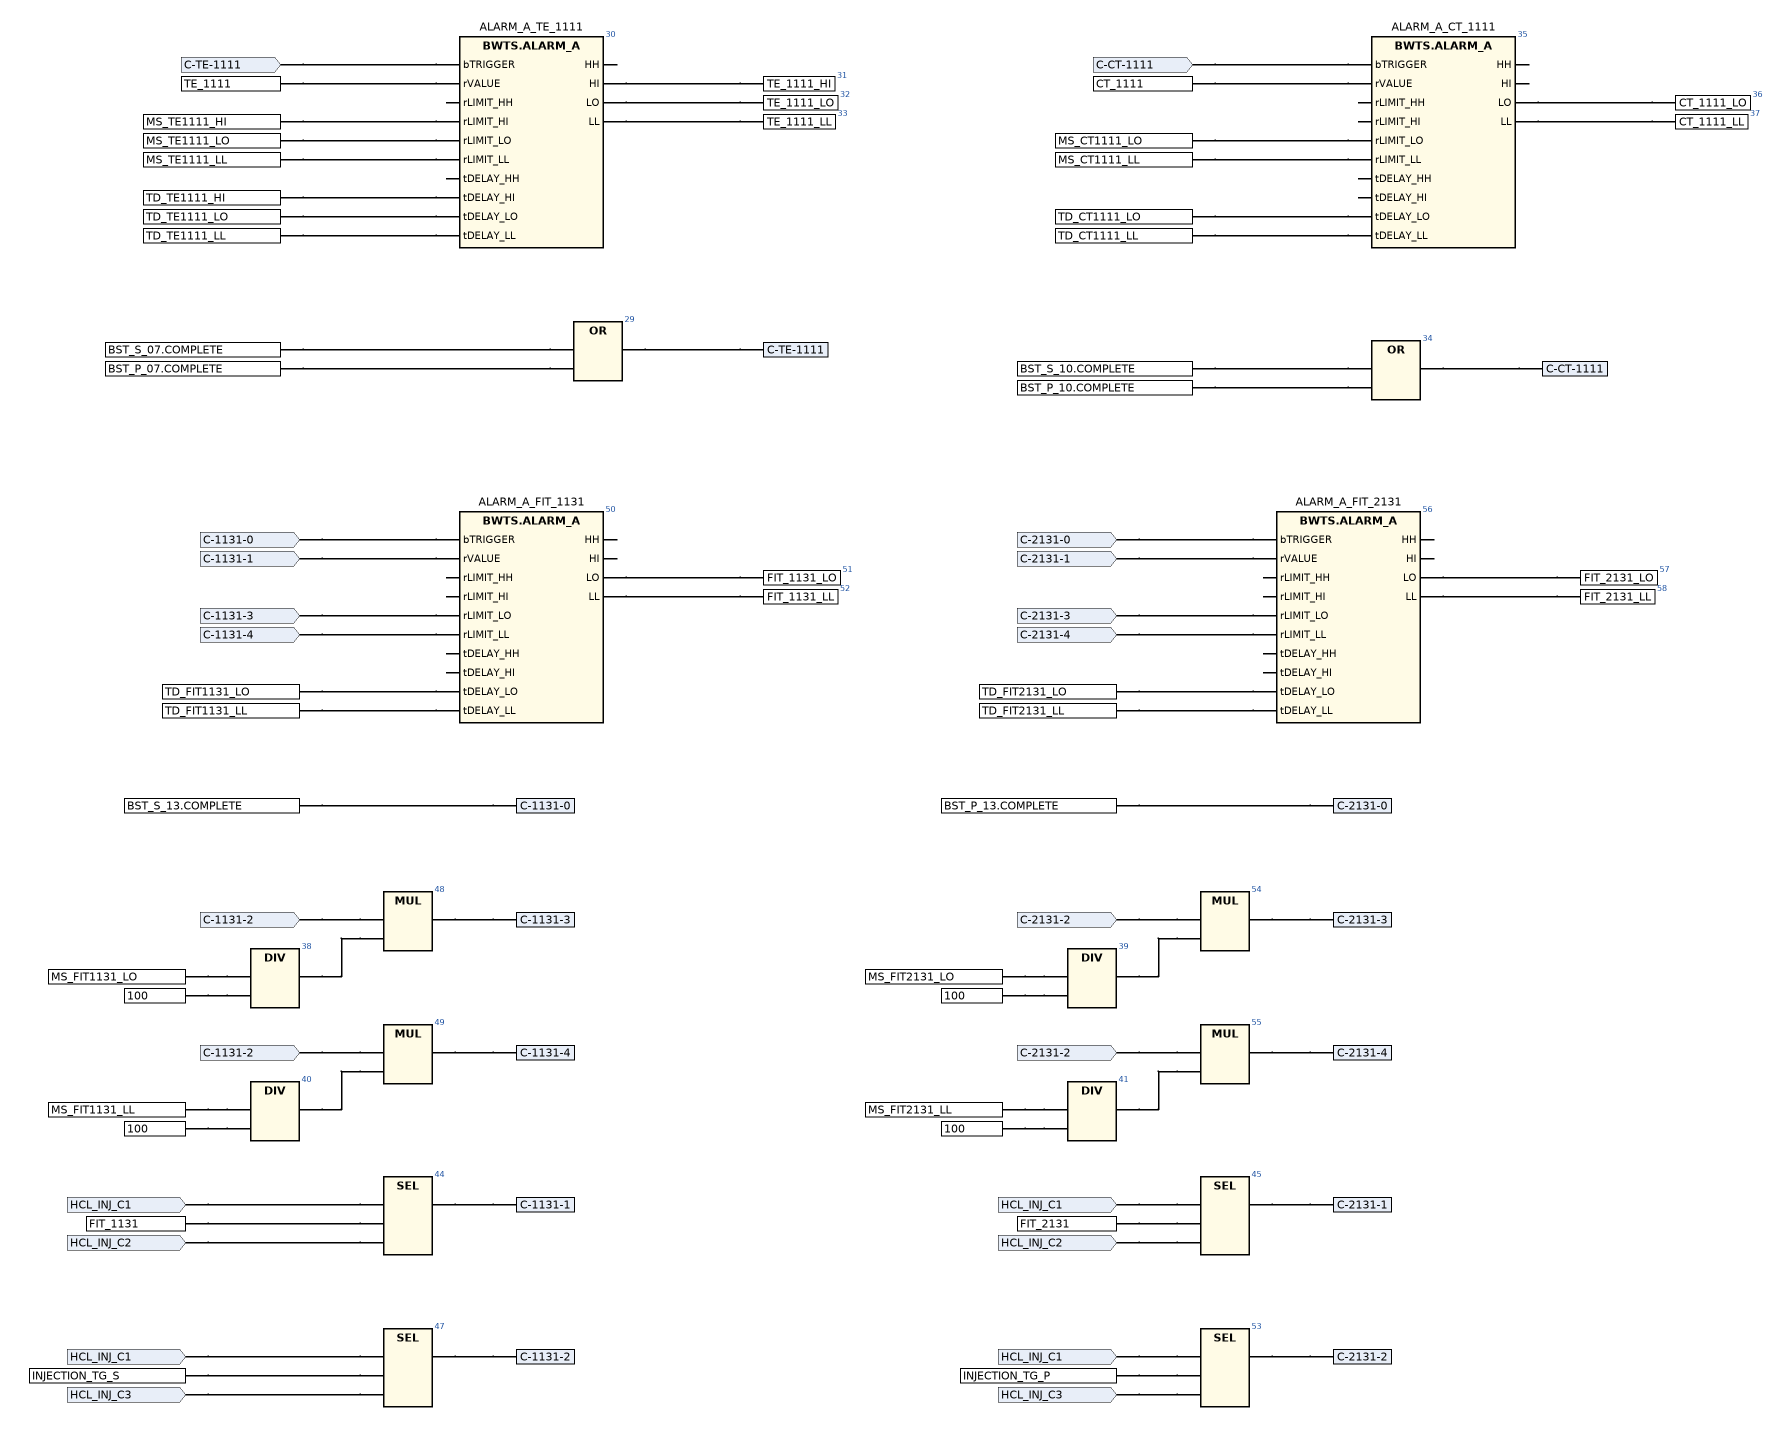
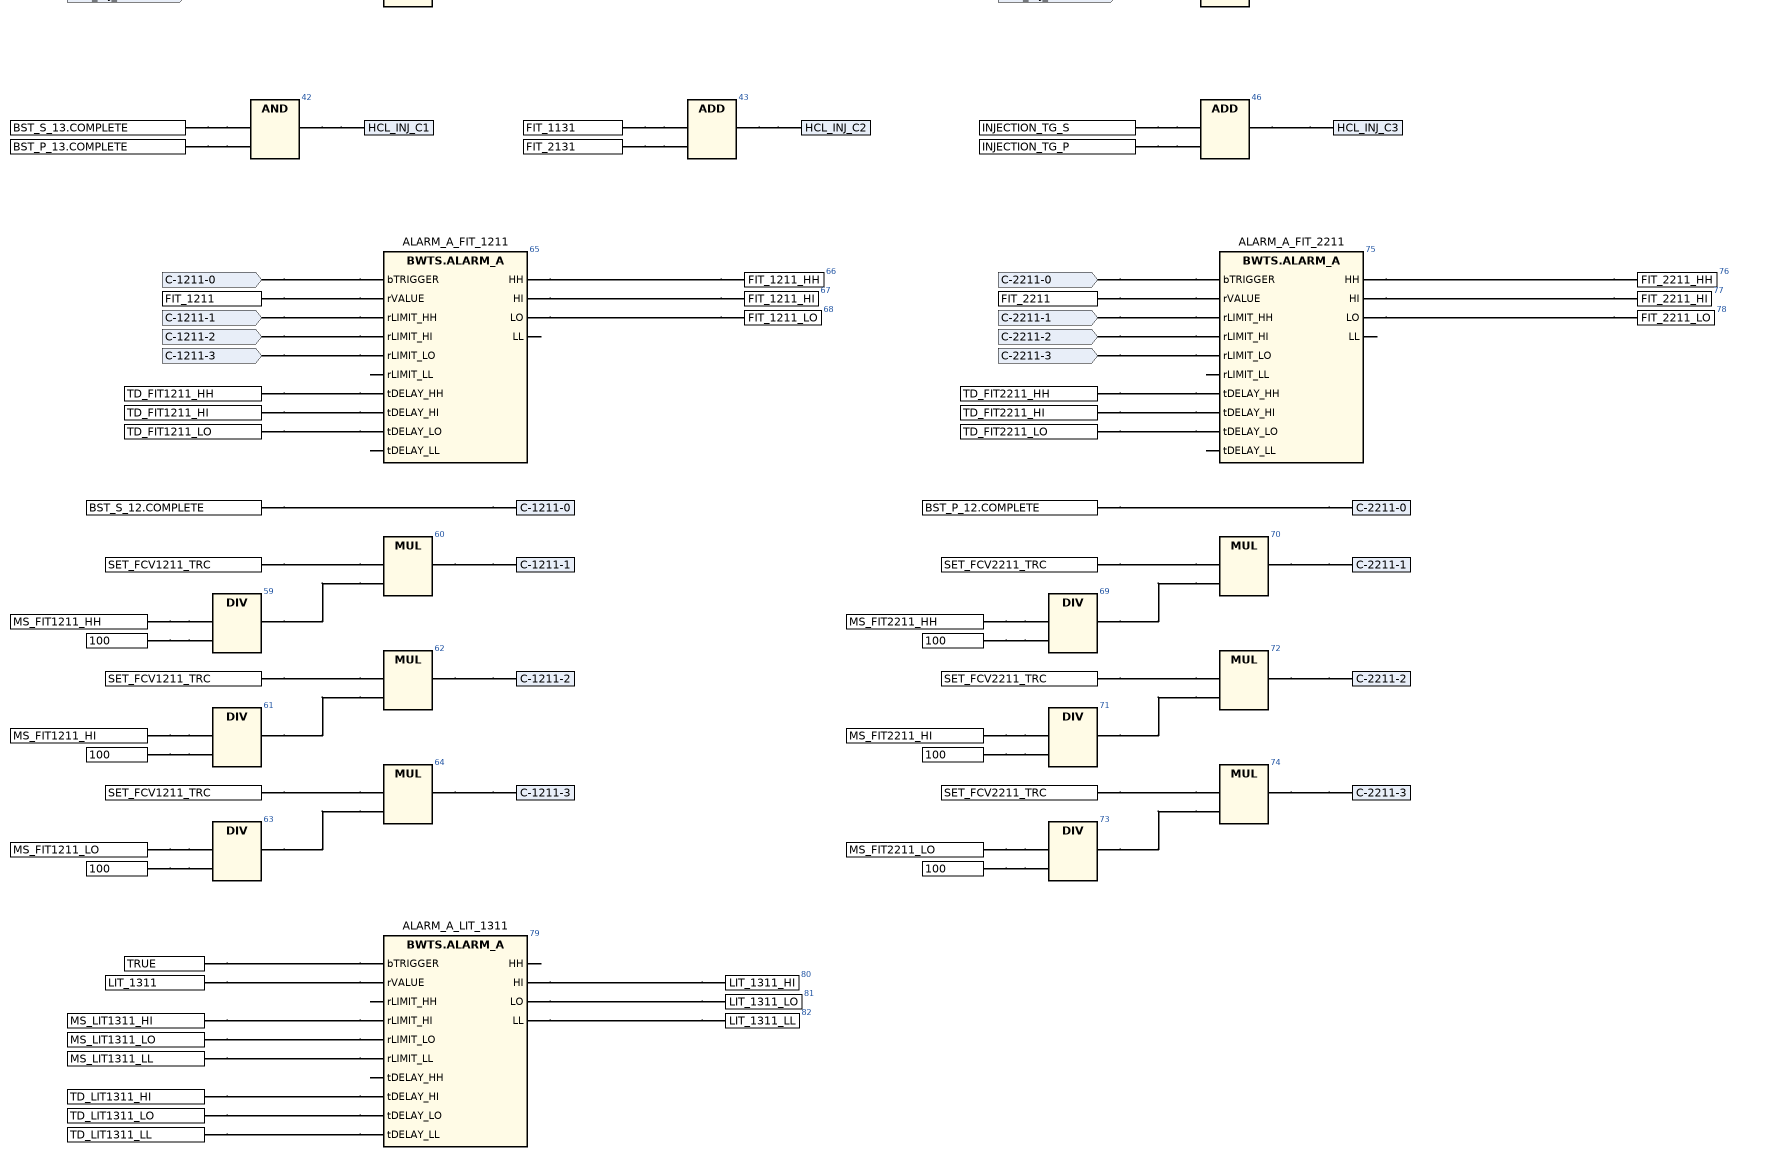
(* BST_S_06.COMPLETE OR BST_P_06.COMPLETE; result not used *)
ALARM_A_PT_1722(
    bTRIGGER := _w1,
    rVALUE := PT_1722,
    rLIMIT_HH := MS_PT1722_HH,
    rLIMIT_HI := MS_PT1722_HI,
    rLIMIT_LO := MS_PT1722_LO,
    tDELAY_HH := TD_PT1722_HH,
    tDELAY_HI := TD_PT1722_HI,
    tDELAY_LO := TD_PT1722_LO); // BWTS.ALARM_A
PT_1722_HH := ALARM_A_PT_1722.HH;
PT_1722_HI := ALARM_A_PT_1722.HI;
PT_1722_LO := ALARM_A_PT_1722.LO;
ALARM_A_PT_1721(
    bTRIGGER := _w2,
    rVALUE := PT_1721,
    rLIMIT_HI := MS_PT1721_HI,
    rLIMIT_LO := MS_PT1721_LO,
    rLIMIT_LL := MS_PT1721_LL,
    tDELAY_HI := TD_PT1721_HI,
    tDELAY_LO := TD_PT1721_LO,
    tDELAY_LL := TD_PT1721_LL); // BWTS.ALARM_A
PT_1721_HI := ALARM_A_PT_1721.HI;
PT_1721_LO := ALARM_A_PT_1721.LO;
PT_1721_LL := ALARM_A_PT_1721.LL;
ALARM_A_P_171(
    bTRIGGER := _w3,
    rVALUE := DP_P171,
    rLIMIT_HH := MS_DP171_HH,
    rLIMIT_HI := MS_DP171_HI,
    tDELAY_HH := TD_DP171_HH,
    tDELAY_HI := TD_DP171_HI); // BWTS.ALARM_A
SWFU_DP_HH := ALARM_A_P_171.HH;
SWFU_DP_HI := ALARM_A_P_171.HI;
(* BST_S_01.COMPLETE OR BST_P_01.COMPLETE; result not used *)
ALARM_A_PT_1121(
    bTRIGGER := _w4,
    rVALUE := PT_1121,
    rLIMIT_HI := MS_PT1121_HI,
    rLIMIT_LO := MS_PT1121_LO,
    rLIMIT_LL := MS_PT1121_LL,
    tDELAY_HI := TD_PT1121_HI,
    tDELAY_LO := TD_PT1121_LO,
    tDELAY_LL := TD_PT1121_LL); // BWTS.ALARM_A
PT_1121_HI := ALARM_A_PT_1121.HI;
PT_1121_LO := ALARM_A_PT_1121.LO;
PT_1121_LL := ALARM_A_PT_1121.LL;
ALARM_A_AIT_1121(
    bTRIGGER := TRUE,
    rVALUE := AIT_1121,
    rLIMIT_HH := MS_AIT1121_HH,
    rLIMIT_HI := MS_AIT1121_HI,
    tDELAY_HH := TD_AIT1121_HH,
    tDELAY_HI := TD_AIT1121_HI); // BWTS.ALARM_A
AIT_1121_HH := ALARM_A_AIT_1121.HH;
AIT_1121_HI := ALARM_A_AIT_1121.HI;
ALARM_A_AIT_1122(
    bTRIGGER := TRUE,
    rVALUE := AIT_1122,
    rLIMIT_HH := MS_AIT1122_HH,
    rLIMIT_HI := MS_AIT1122_HI,
    tDELAY_HH := TD_AIT1122_HH,
    tDELAY_HI := TD_AIT1122_HI); // BWTS.ALARM_A
AIT_1122_HH := ALARM_A_AIT_1122.HH;
AIT_1122_HI := ALARM_A_AIT_1122.HI;
ALARM_A_AIT_1123(
    bTRIGGER := TRUE,
    rVALUE := AIT_1123,
    rLIMIT_HH := MS_AIT1123_HH,
    rLIMIT_HI := MS_AIT1123_HI,
    tDELAY_HH := TD_AIT1123_HH,
    tDELAY_HI := TD_AIT1123_HI); // BWTS.ALARM_A
AIT_1123_HH := ALARM_A_AIT_1123.HH;
AIT_1123_HI := ALARM_A_AIT_1123.HI;
ALARM_A_AP_LVL_01(
    bTRIGGER := MF_APT,
    rVALUE := AP_LVL_01,
    rLIMIT_LO := MS_AP_LO,
    rLIMIT_LL := MS_AP_LL,
    tDELAY_LO := TD_AP_LO,
    tDELAY_LL := TD_AP_LL); // BWTS.ALARM_A
AP_LVL_LO := ALARM_A_AP_LVL_01.LO;
AP_LVL_LL := ALARM_A_AP_LVL_01.LL;
(* BST_S_07.COMPLETE OR BST_P_07.COMPLETE; result not used *)
ALARM_A_TE_1111(
    bTRIGGER := _w5,
    rVALUE := TE_1111,
    rLIMIT_HI := MS_TE1111_HI,
    rLIMIT_LO := MS_TE1111_LO,
    rLIMIT_LL := MS_TE1111_LL,
    tDELAY_HI := TD_TE1111_HI,
    tDELAY_LO := TD_TE1111_LO,
    tDELAY_LL := TD_TE1111_LL); // BWTS.ALARM_A
TE_1111_HI := ALARM_A_TE_1111.HI;
TE_1111_LO := ALARM_A_TE_1111.LO;
TE_1111_LL := ALARM_A_TE_1111.LL;
(* BST_S_10.COMPLETE OR BST_P_10.COMPLETE; result not used *)
ALARM_A_CT_1111(
    bTRIGGER := _w6,
    rVALUE := CT_1111,
    rLIMIT_LO := MS_CT1111_LO,
    rLIMIT_LL := MS_CT1111_LL,
    tDELAY_LO := TD_CT1111_LO,
    tDELAY_LL := TD_CT1111_LL); // BWTS.ALARM_A
CT_1111_LO := ALARM_A_CT_1111.LO;
CT_1111_LL := ALARM_A_CT_1111.LL;
_w7 := MS_FIT2131_LO / 100;
_w8 := MS_FIT2131_LL / 100;
(* BST_S_13.COMPLETE AND BST_P_13.COMPLETE; result not used *)
(* FIT_1131 + FIT_2131; result not used *)
(* SEL(_w9, FIT_1131, _w10); result not used *)
(* SEL(_w11, FIT_2131, _w12); result not used *)
(* INJECTION_TG_S + INJECTION_TG_P; result not used *)
(* SEL(_w13, INJECTION_TG_S, _w14); result not used *)
(* _w15 * (MS_FIT1131_LO / 100); result not used *)
(* _w16 * (MS_FIT1131_LL / 100); result not used *)
ALARM_A_FIT_1131(
    bTRIGGER := _w17,
    rVALUE := _w18,
    rLIMIT_LO := _w19,
    rLIMIT_LL := _w20,
    tDELAY_LO := TD_FIT1131_LO,
    tDELAY_LL := TD_FIT1131_LL); // BWTS.ALARM_A
FIT_1131_LO := ALARM_A_FIT_1131.LO;
FIT_1131_LL := ALARM_A_FIT_1131.LL;
(* SEL(_w21, INJECTION_TG_P, _w22); result not used *)
(* _w23 * _w7; result not used *)
(* _w24 * _w8; result not used *)
ALARM_A_FIT_2131(
    bTRIGGER := _w25,
    rVALUE := _w26,
    rLIMIT_LO := _w27,
    rLIMIT_LL := _w28,
    tDELAY_LO := TD_FIT2131_LO,
    tDELAY_LL := TD_FIT2131_LL); // BWTS.ALARM_A
FIT_2131_LO := ALARM_A_FIT_2131.LO;
FIT_2131_LL := ALARM_A_FIT_2131.LL;
(* SET_FCV1211_TRC * (MS_FIT1211_HH / 100); result not used *)
(* SET_FCV1211_TRC * (MS_FIT1211_HI / 100); result not used *)
(* SET_FCV1211_TRC * (MS_FIT1211_LO / 100); result not used *)
ALARM_A_FIT_1211(
    bTRIGGER := _w29,
    rVALUE := FIT_1211,
    rLIMIT_HH := _w30,
    rLIMIT_HI := _w31,
    rLIMIT_LO := _w32,
    tDELAY_HH := TD_FIT1211_HH,
    tDELAY_HI := TD_FIT1211_HI,
    tDELAY_LO := TD_FIT1211_LO); // BWTS.ALARM_A
FIT_1211_HH := ALARM_A_FIT_1211.HH;
FIT_1211_HI := ALARM_A_FIT_1211.HI;
FIT_1211_LO := ALARM_A_FIT_1211.LO;
(* SET_FCV2211_TRC * (MS_FIT2211_HH / 100); result not used *)
(* SET_FCV2211_TRC * (MS_FIT2211_HI / 100); result not used *)
(* SET_FCV2211_TRC * (MS_FIT2211_LO / 100); result not used *)
ALARM_A_FIT_2211(
    bTRIGGER := _w33,
    rVALUE := FIT_2211,
    rLIMIT_HH := _w34,
    rLIMIT_HI := _w35,
    rLIMIT_LO := _w36,
    tDELAY_HH := TD_FIT2211_HH,
    tDELAY_HI := TD_FIT2211_HI,
    tDELAY_LO := TD_FIT2211_LO); // BWTS.ALARM_A
FIT_2211_HH := ALARM_A_FIT_2211.HH;
FIT_2211_HI := ALARM_A_FIT_2211.HI;
FIT_2211_LO := ALARM_A_FIT_2211.LO;
ALARM_A_LIT_1311(
    bTRIGGER := TRUE,
    rVALUE := LIT_1311,
    rLIMIT_HI := MS_LIT1311_HI,
    rLIMIT_LO := MS_LIT1311_LO,
    rLIMIT_LL := MS_LIT1311_LL,
    tDELAY_HI := TD_LIT1311_HI,
    tDELAY_LO := TD_LIT1311_LO,
    tDELAY_LL := TD_LIT1311_LL); // BWTS.ALARM_A
LIT_1311_HI := ALARM_A_LIT_1311.HI;
LIT_1311_LO := ALARM_A_LIT_1311.LO;
LIT_1311_LL := ALARM_A_LIT_1311.LL;

END_PROGRAM

// Device/Application/Logic/0.ALARM/ALARM_INTERLOCK_D_1
PROGRAM ALARM_INTERLOCK_D_1
VAR
	//Library
	ALARM_D_CC_ESTOP,
	ALARM_D_HMI_ESTOP,
	ALARM_D_RF_ESTOP,
	ALARM_D_CC_TEMP,
	ALARM_D_MCC_OFF,
	ALARM_D_B117A_OFF,
	ALARM_D_B117B_OFF,
	ALARM_D_P171A_OFF,
	ALARM_D_P171B_OFF,
	ALARM_D_B117A_F,
	ALARM_D_B117B_F,
	ALARM_D_P171A_F,
	ALARM_D_P171B_F,	
	ALARM_D_P132_TRIP,
	ALARM_D_P232_TRIP,
	
	ALARM_D_RF142A_E,
	ALARM_D_RF142B_E,
	ALARM_D_RF142C_E,
	ALARM_D_COUPLER_E,
	ALARM_D_BLR_SPD,
	ALARM_D_SWP_SPD,
	ALARM_D_RF_SPD,
	ALARM_D_LS_1111,
	ALARM_D_LS_1141,
	ALARM_D_ZS_1112A_CL,
	ALARM_D_ZS_1113A_CL,
	ALARM_D_ZS_1114A_CL,
	ALARM_D_ZS_1112A_OP,
	ALARM_D_ZS_1113A_OP,
	ALARM_D_ZS_1114A_OP,
	ALARM_D_WBP_01_AL,
	ALARM_D_WBP_02_AL,
	ALARM_D_WBP_01_FAULT,
	ALARM_D_WBP_02_FAULT,
	ALARM_D_GSP_01_AL,
	ALARM_D_GSP_02_AL,
	ALARM_D_GSP_01_FAULT,
	ALARM_D_GSP_02_FAULT,
	ALARM_D_DPS_1321,
	ALARM_D_DPS_2321,
	ALARM_D_RFS_1131,
	ALARM_D_RFS_2131,
	ALARM_D_AIT_151_E,
	ALARM_D_AIT_151_F,
	ALARM_D_AIT_251_E,
	ALARM_D_AIT_251_F,
	
	ALARM_D_BLR_BYPASS,
	ALARM_D_LS_1901_HH,
	
	ALARM_D_GAS_LEAK_AL
	: BWTS.ALARM_D;
	TON_AIT151_E: TON;
	TON_AIT151_F: TON;
	
	TON_AIT251_E: TON;
	TON_AIT251_F: TON;
END_VAR
VAR // added by the converter: edge detectors and wires of the graphical bodies
    _w1, _w2, _w3, _w4, _w5, _w6, _w7, _w8, _w9, _w10, _w11, _w12, _w13, _w14, _w15, _w16, _w17, _w18, _w19, _w20 : ANY;
END_VAR

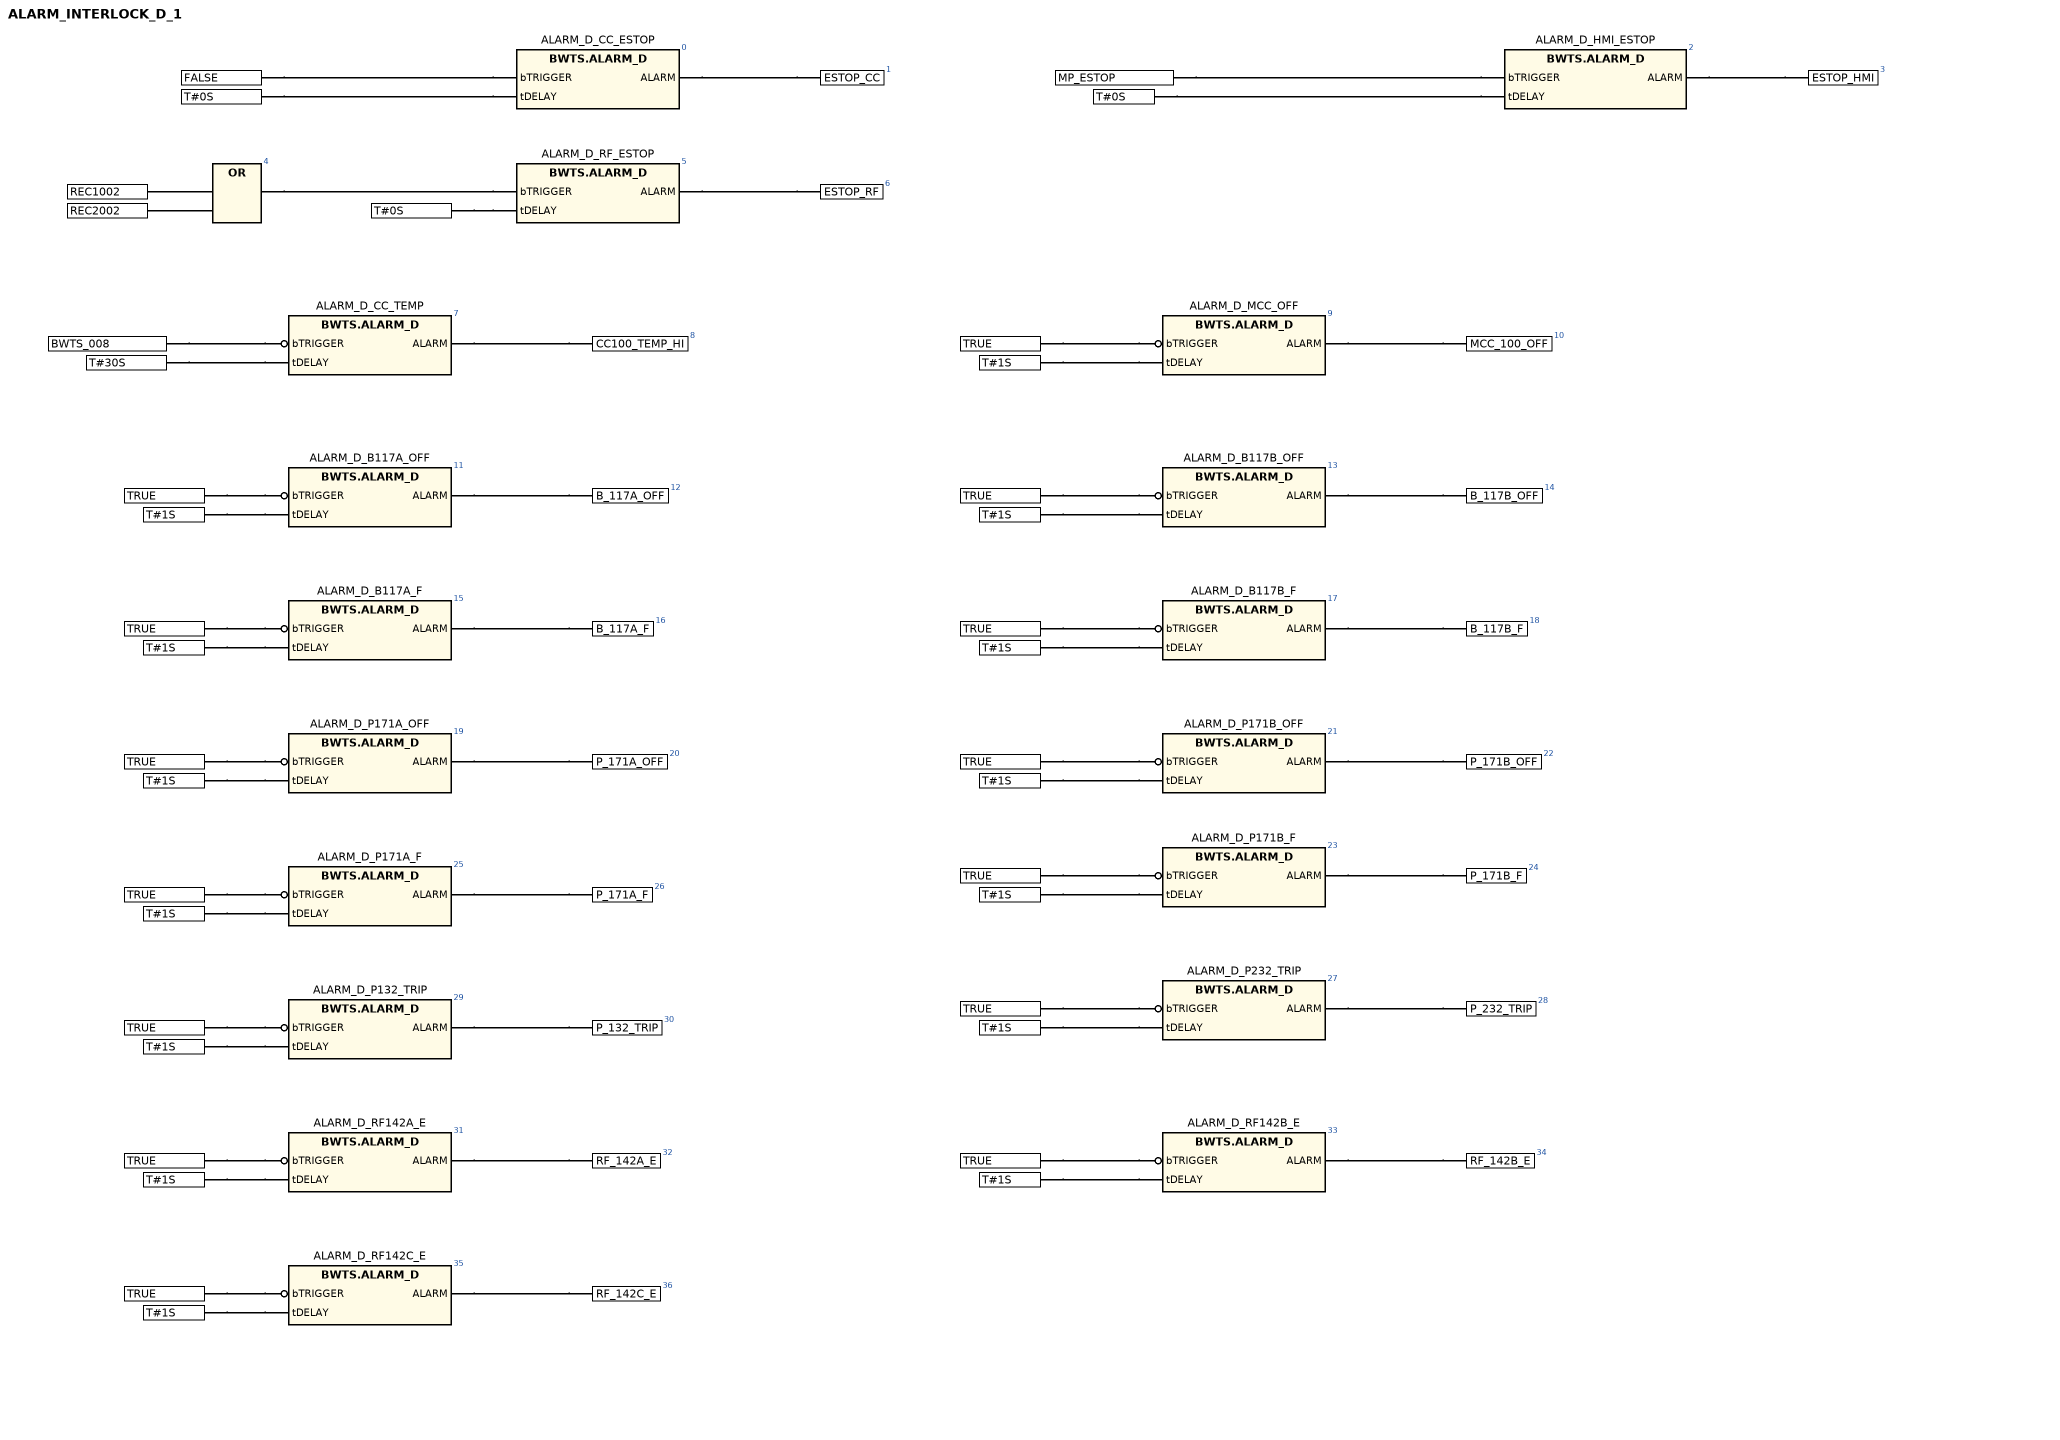
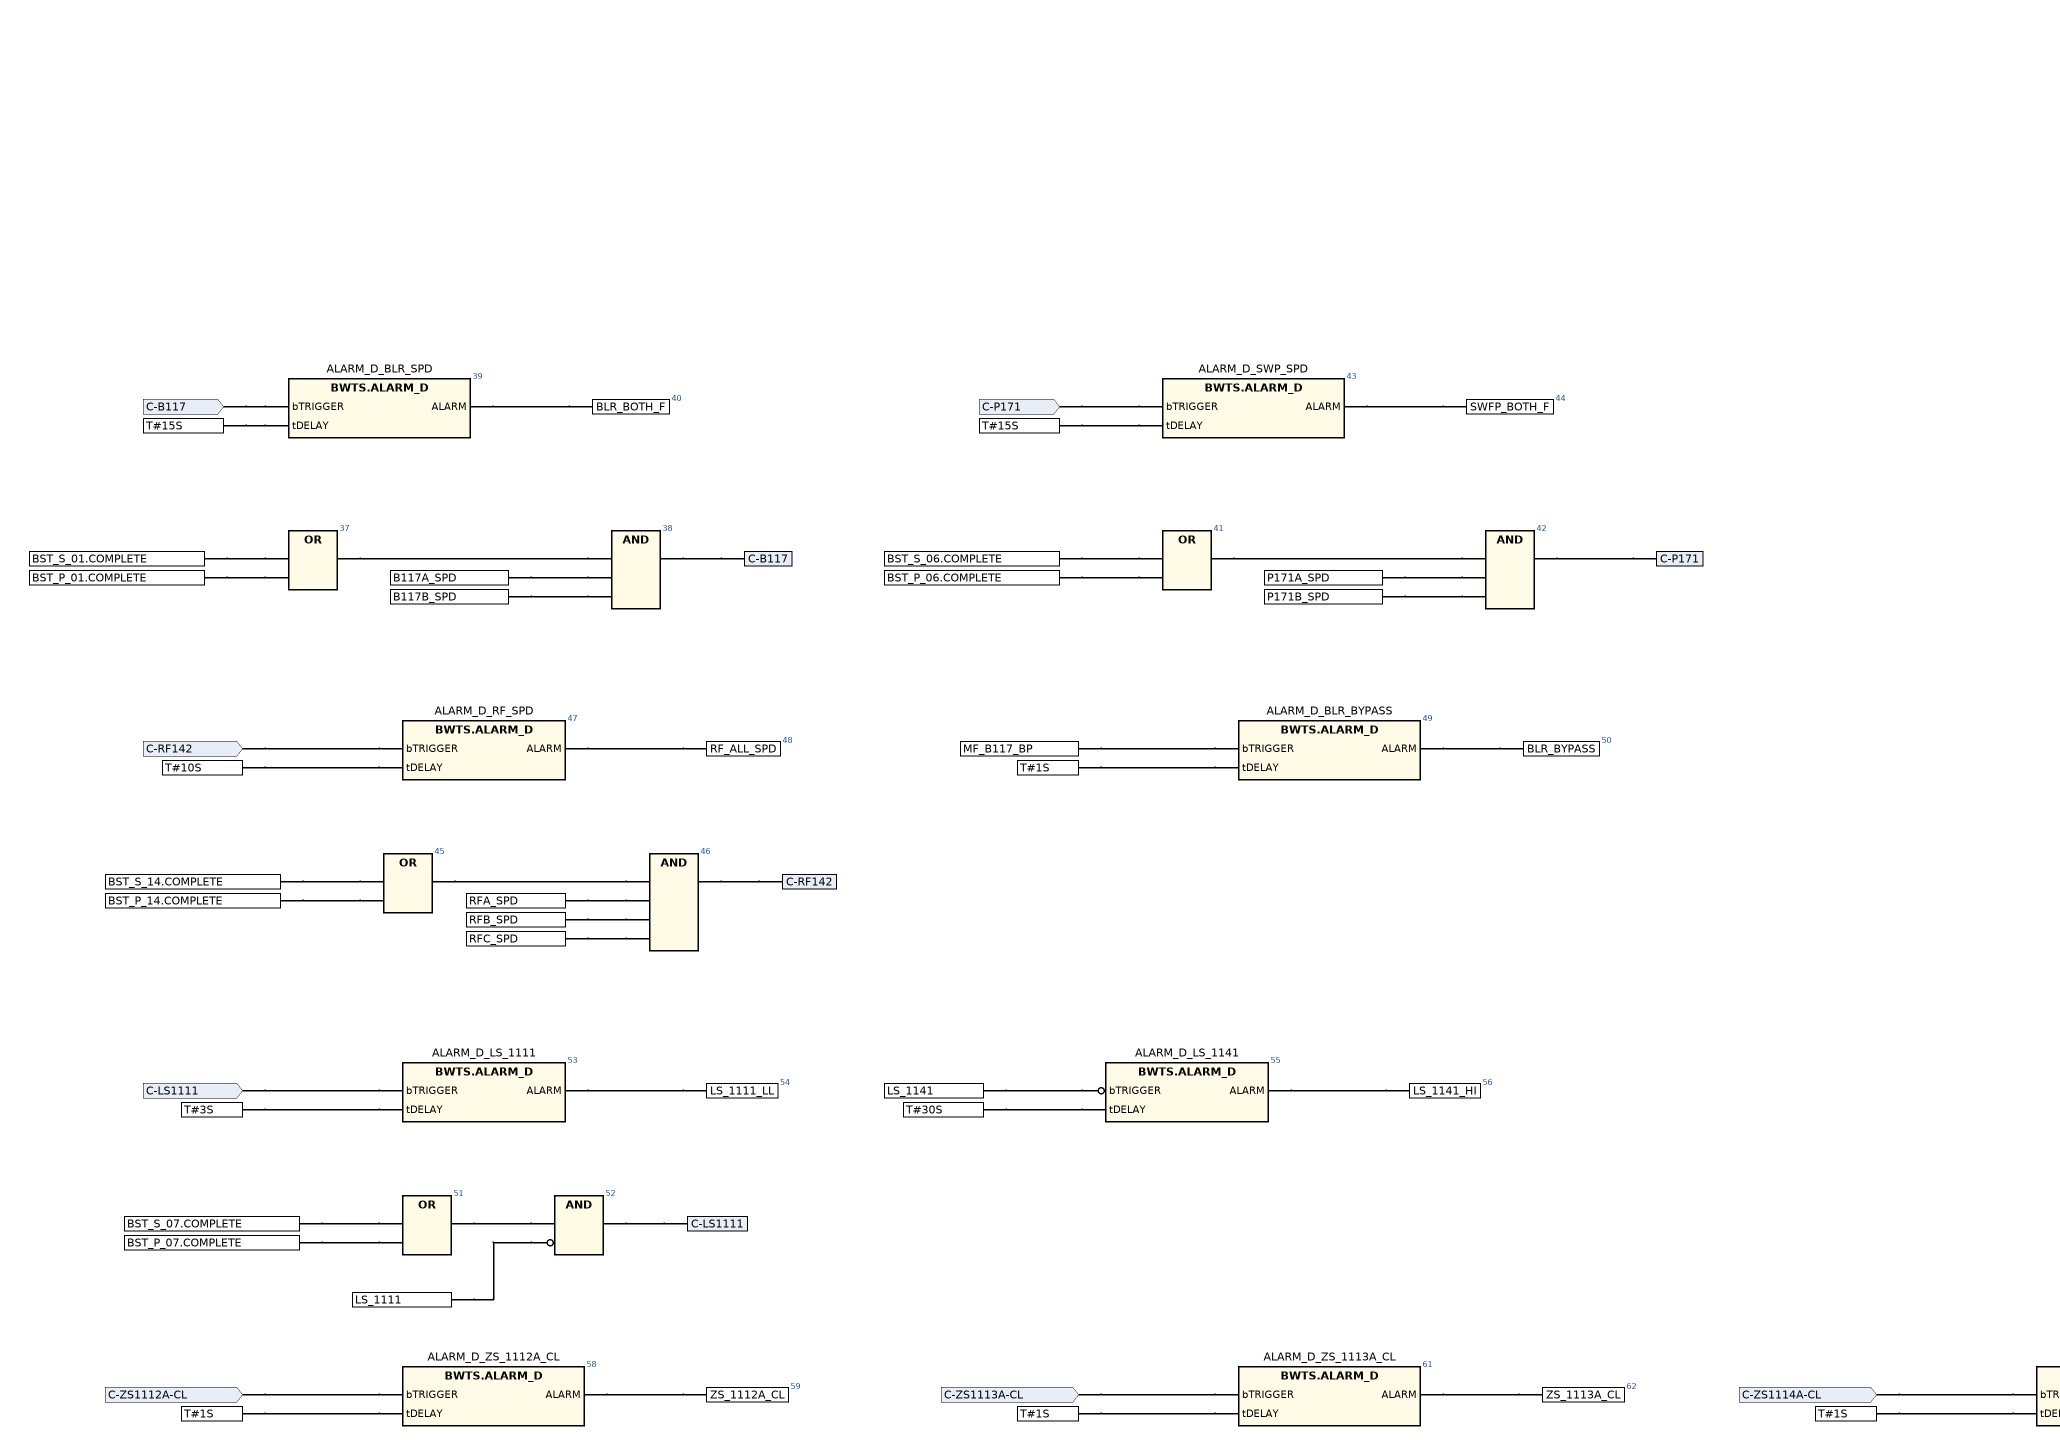
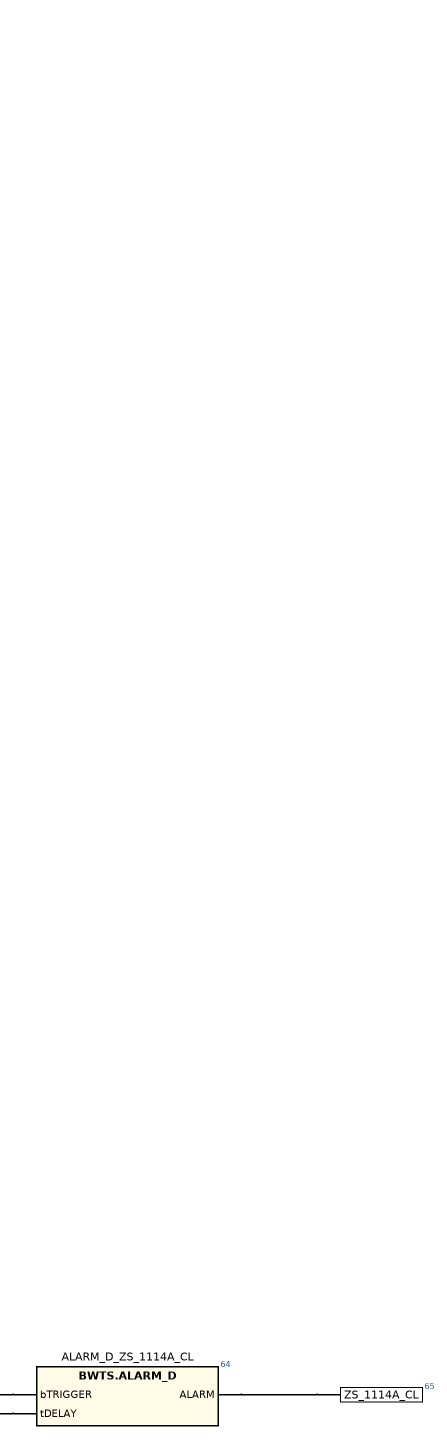
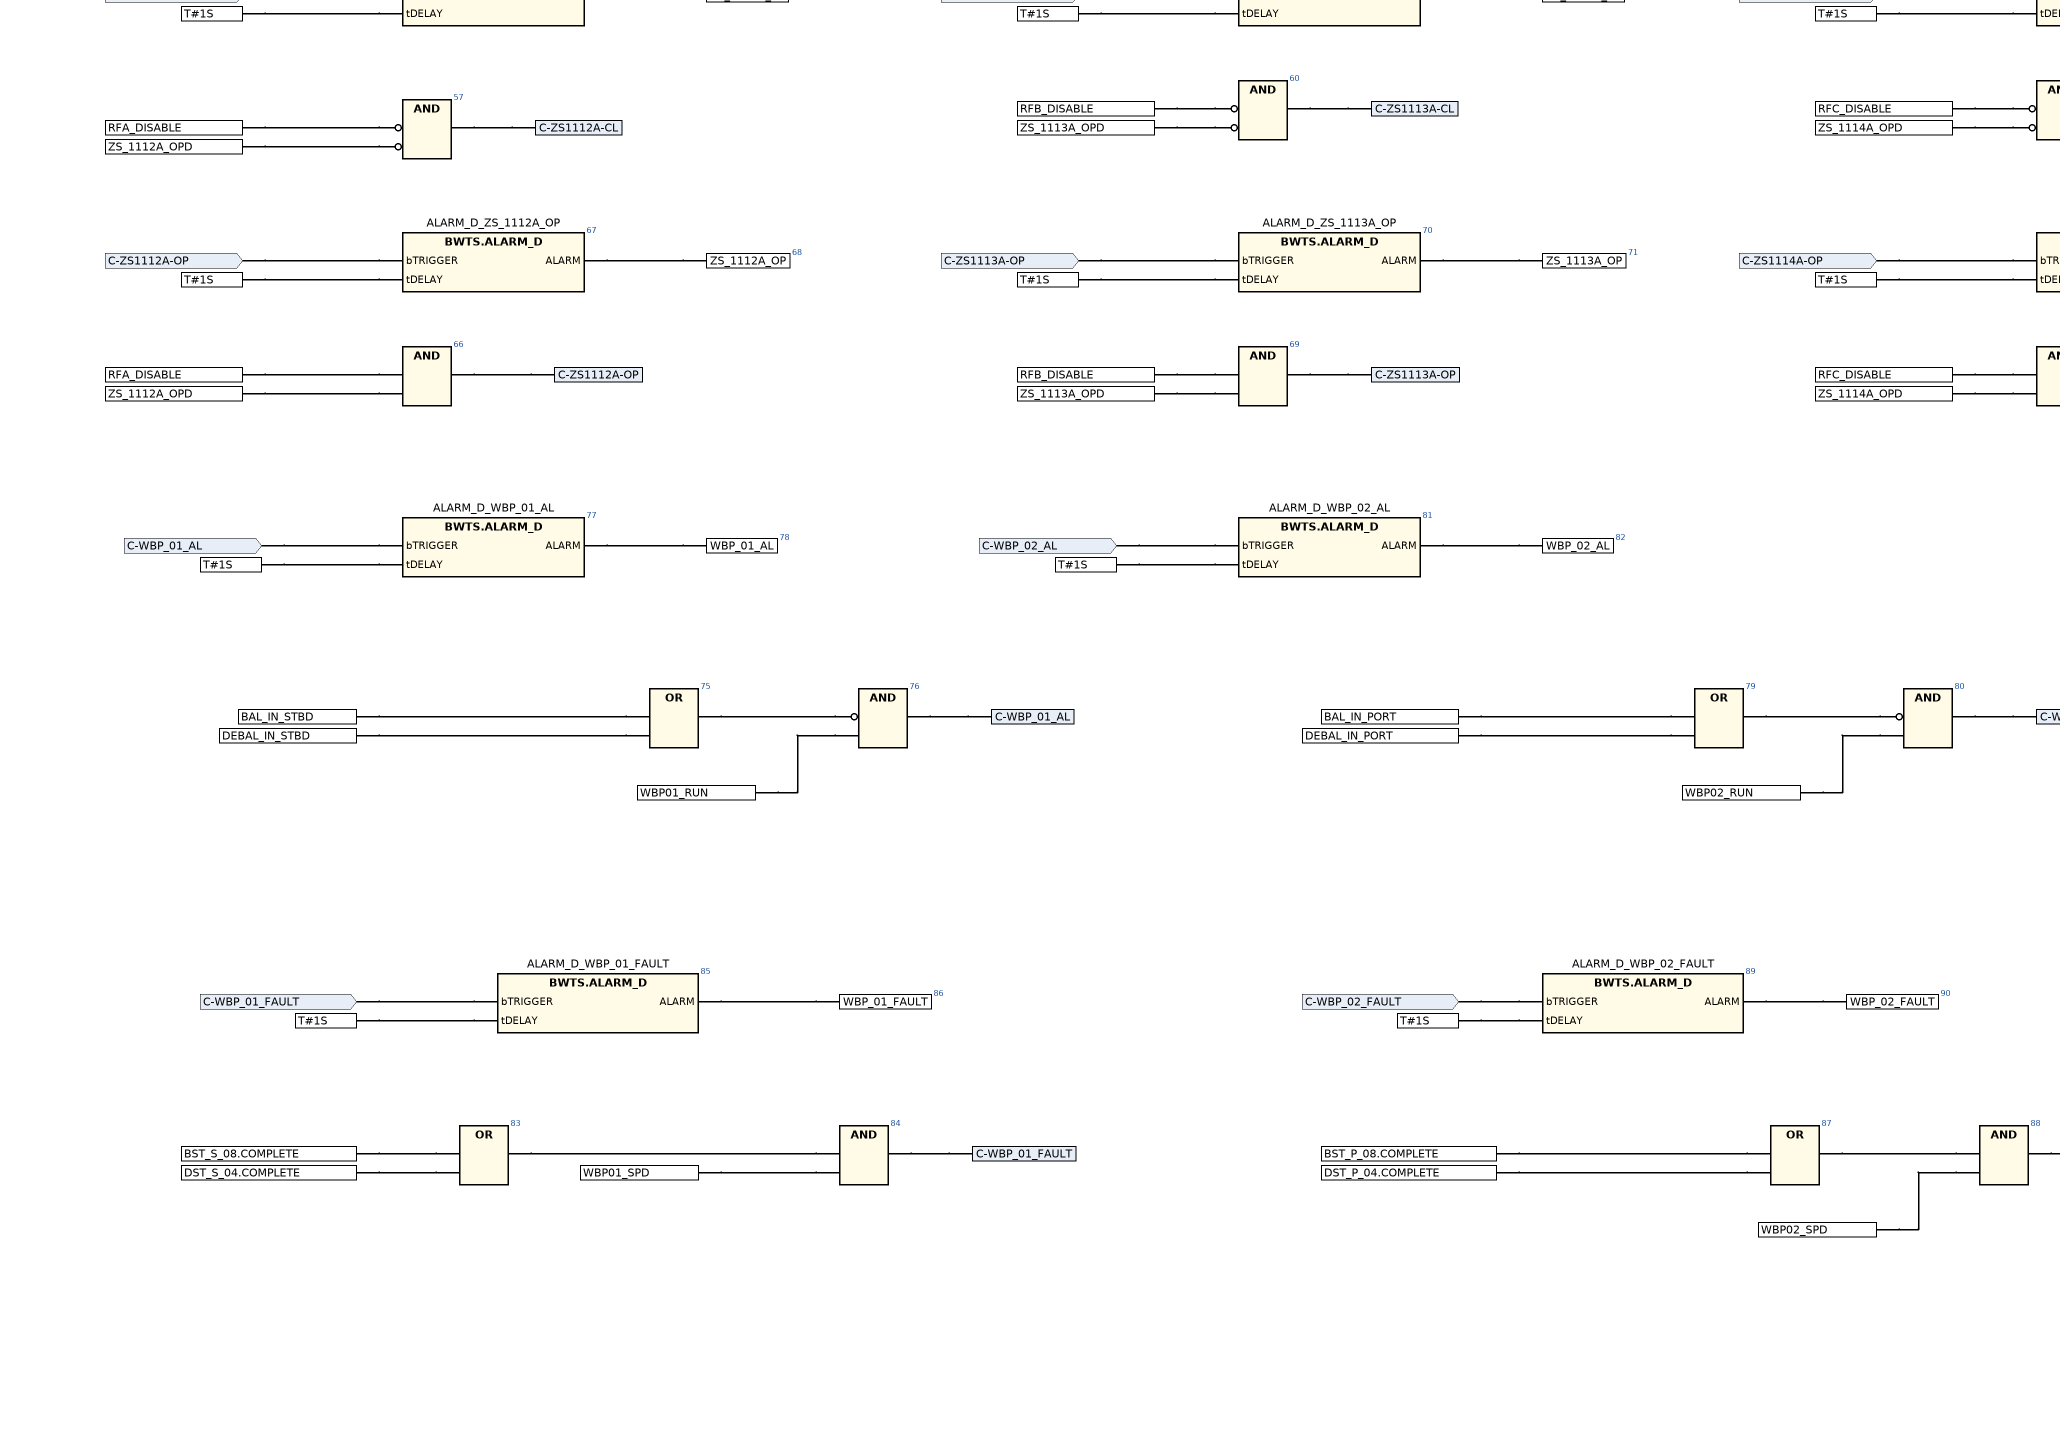
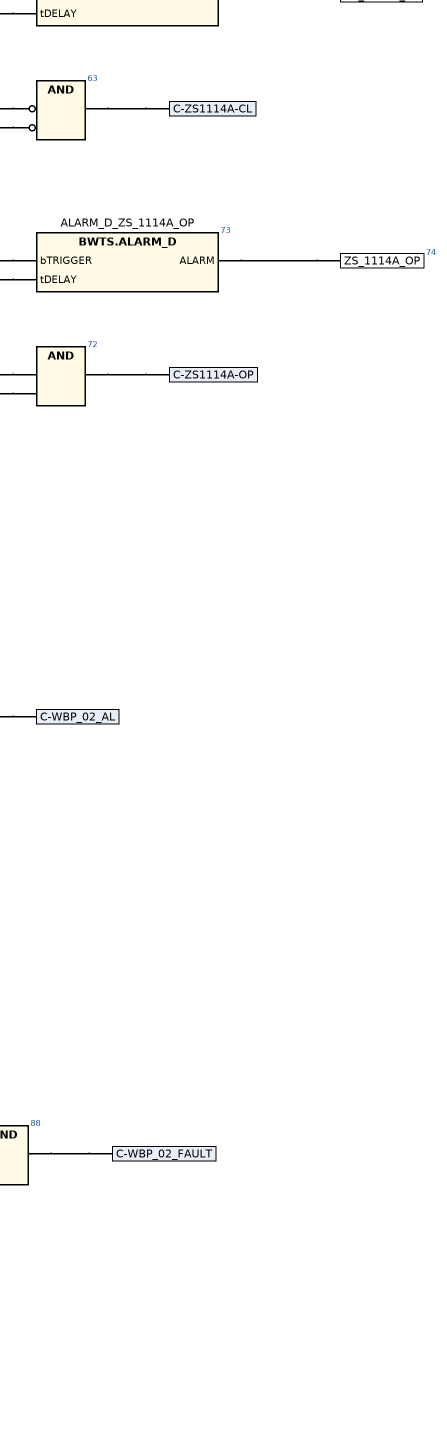
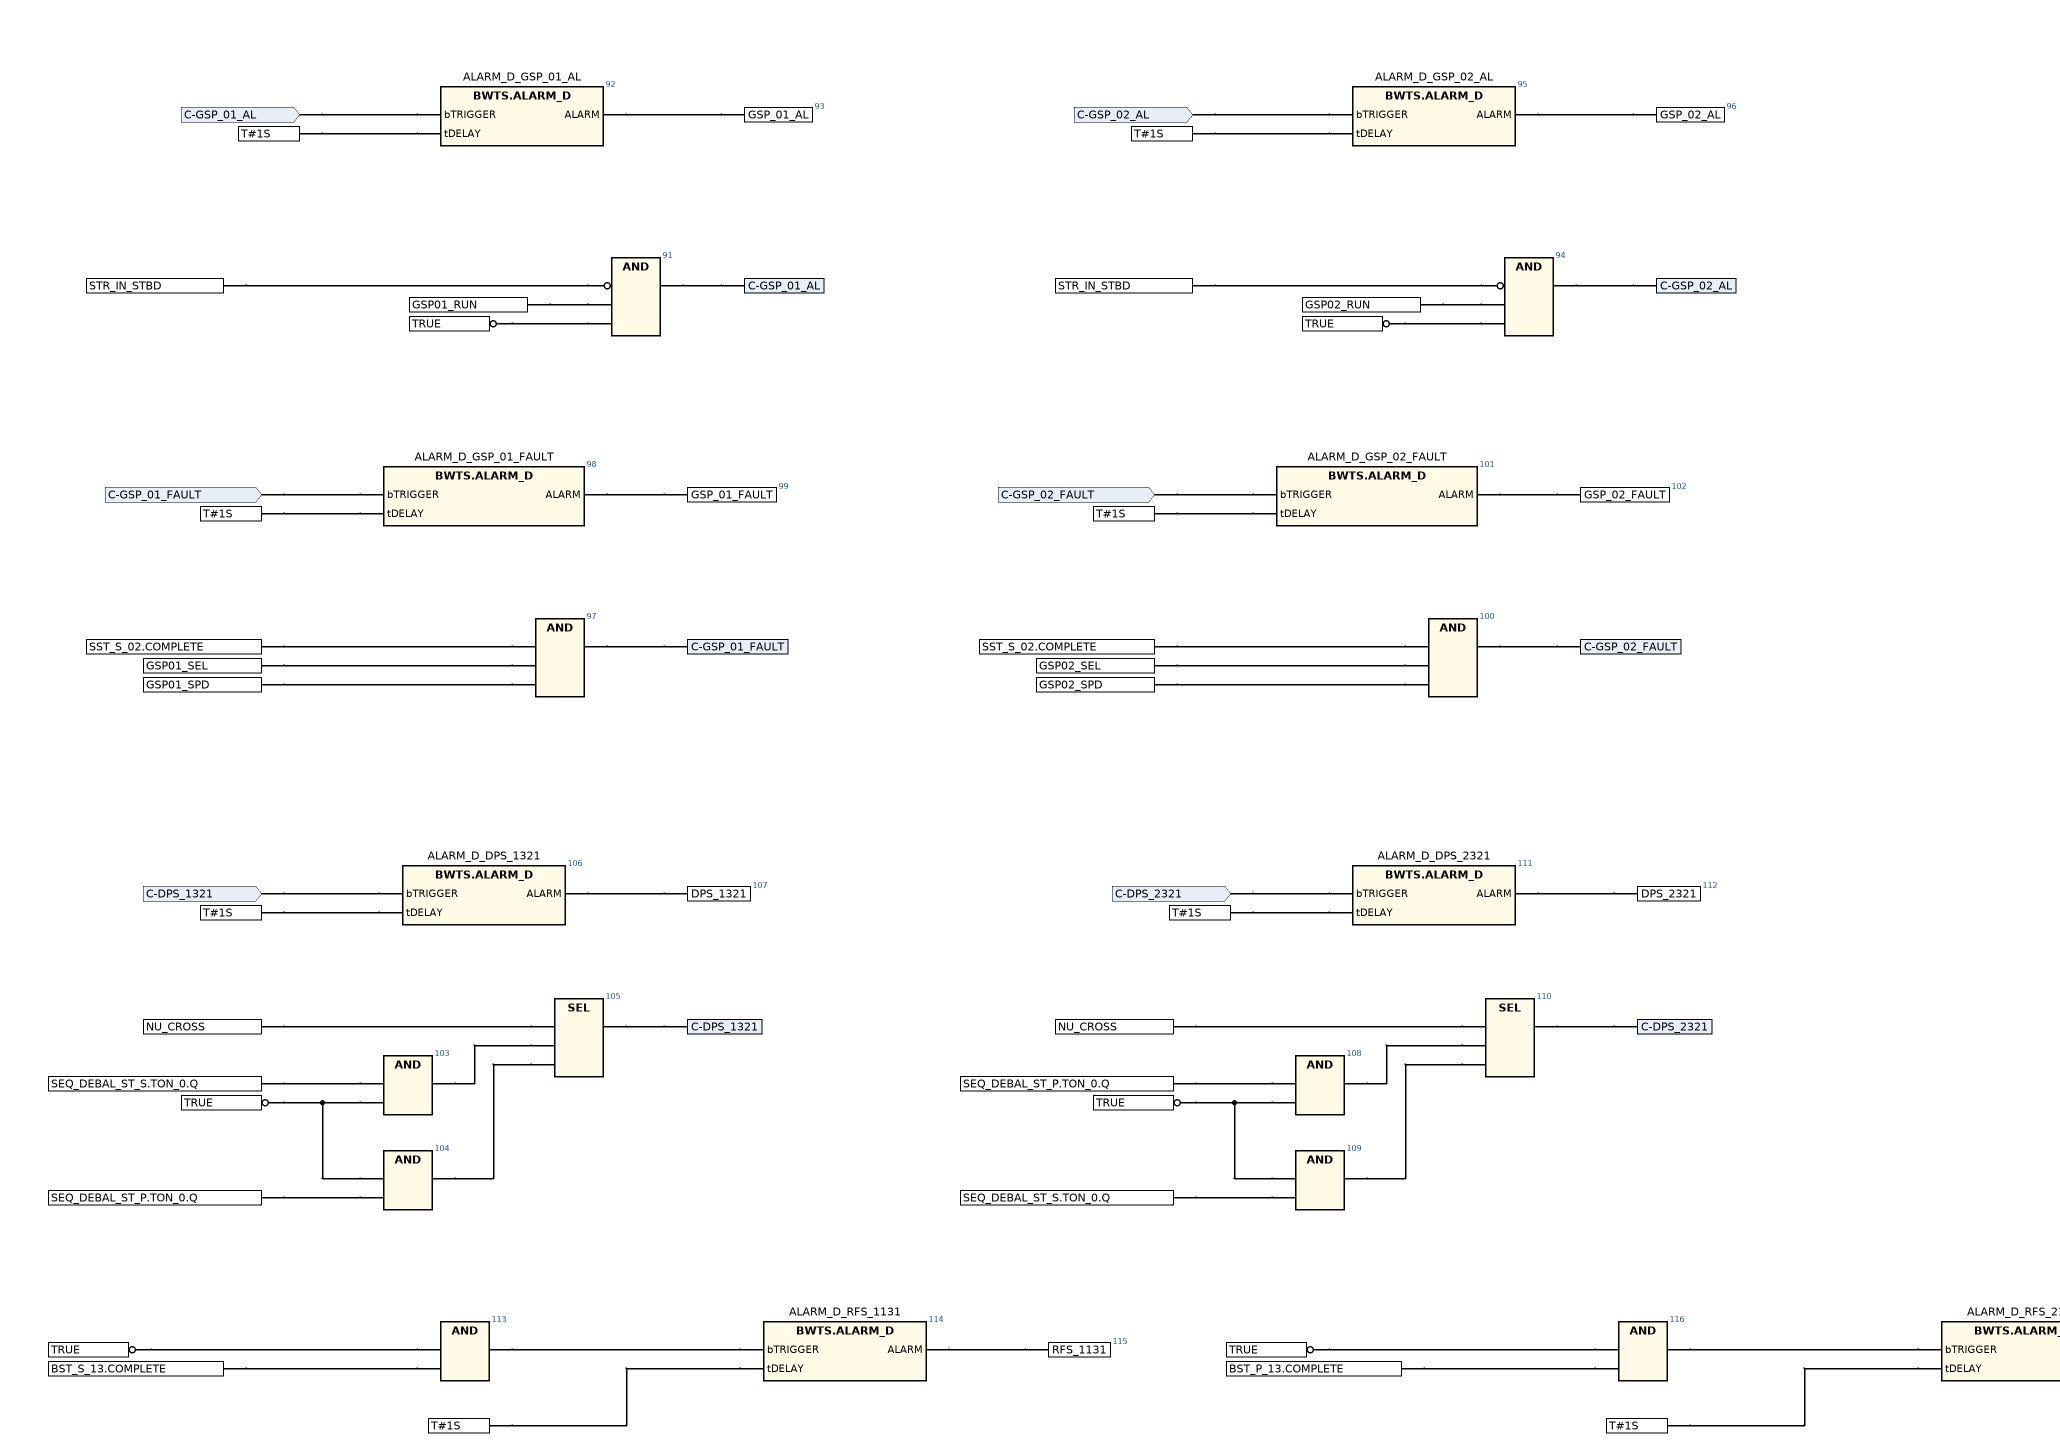
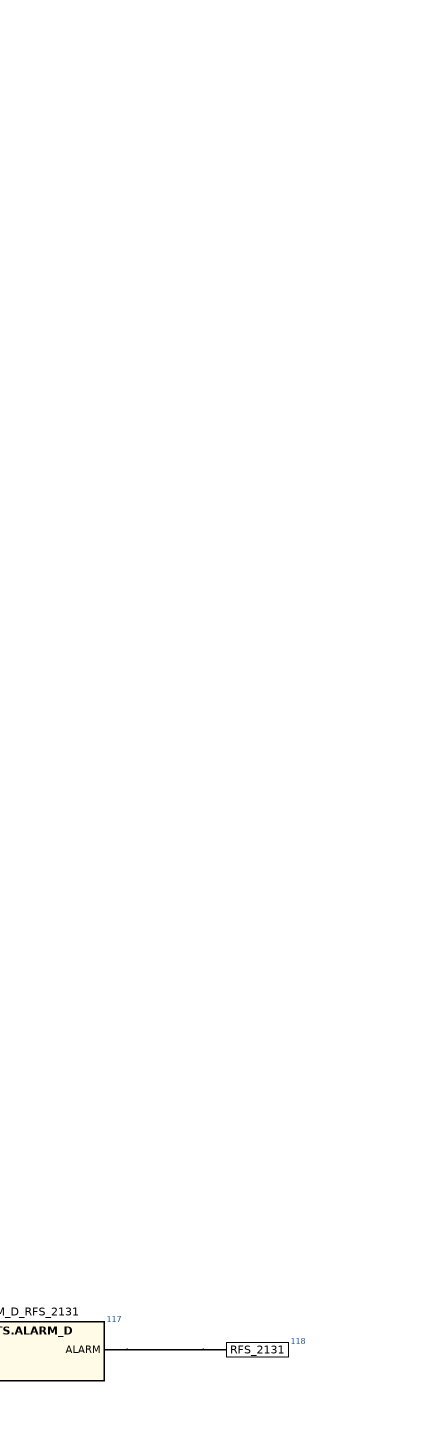
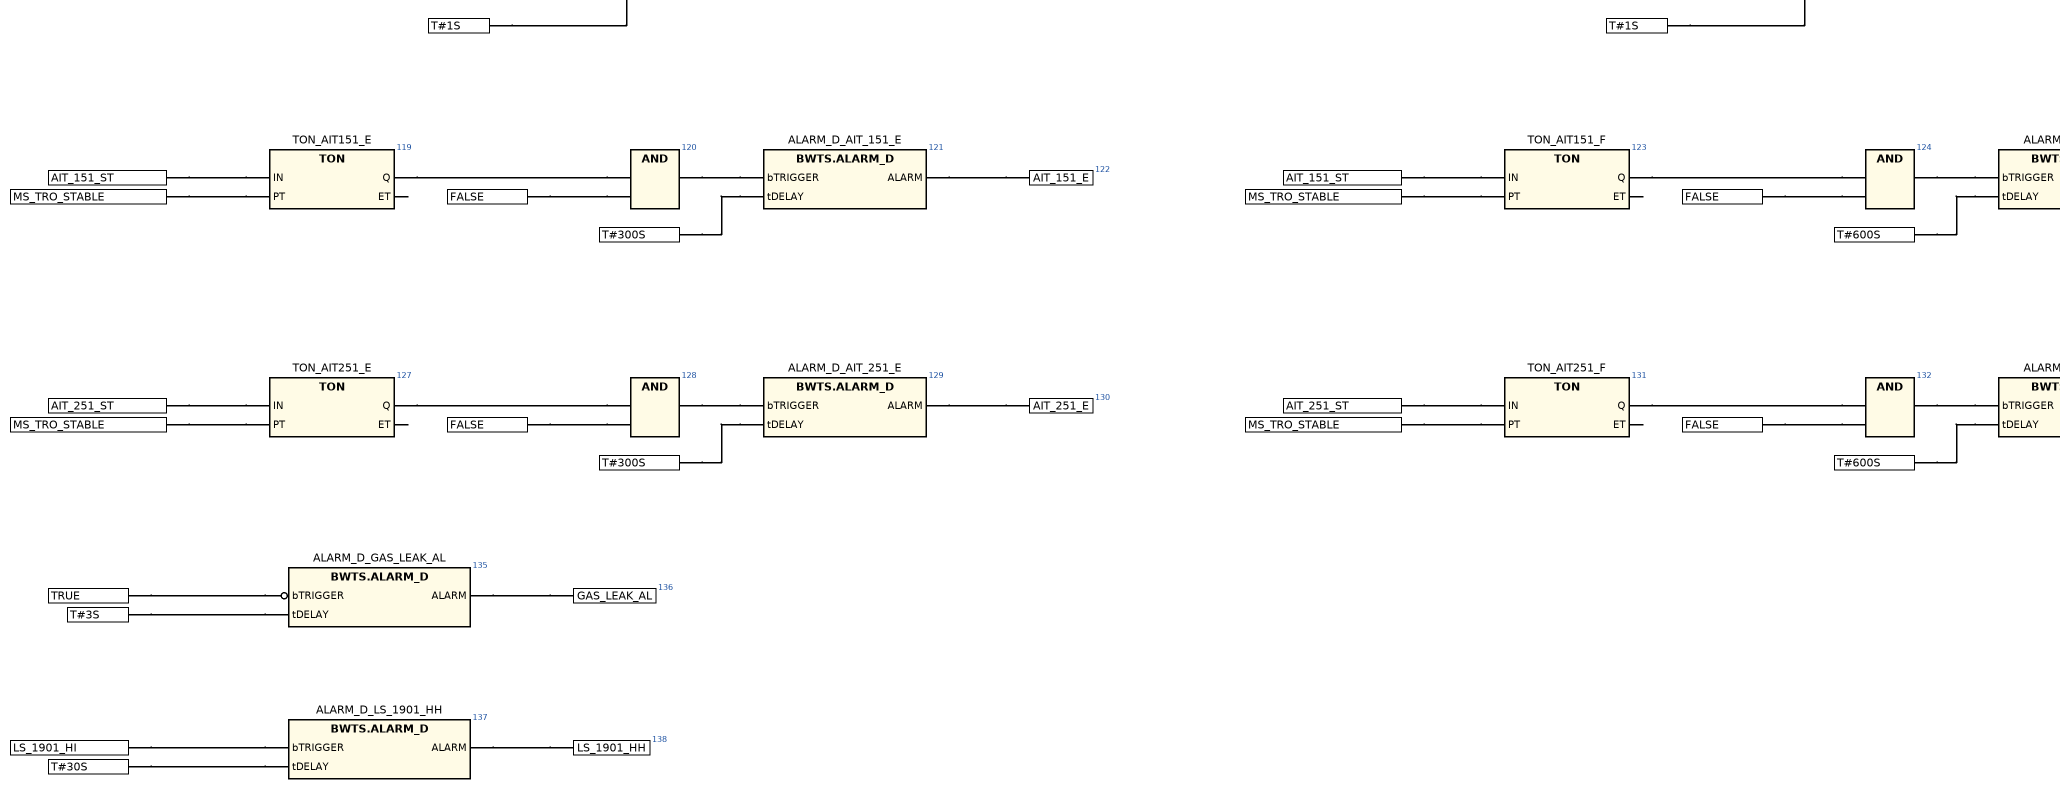
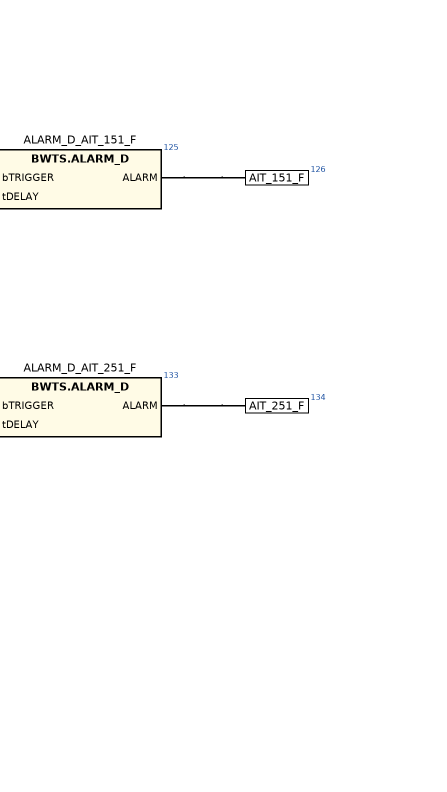
ALARM_D_CC_ESTOP(bTRIGGER := FALSE, tDELAY := T#0S); // BWTS.ALARM_D
ESTOP_CC := ALARM_D_CC_ESTOP.ALARM;
ALARM_D_HMI_ESTOP(bTRIGGER := MP_ESTOP, tDELAY := T#0S); // BWTS.ALARM_D
ESTOP_HMI := ALARM_D_HMI_ESTOP.ALARM;
ALARM_D_RF_ESTOP(bTRIGGER := REC1002 OR REC2002, tDELAY := T#0S); // BWTS.ALARM_D
ESTOP_RF := ALARM_D_RF_ESTOP.ALARM;
ALARM_D_CC_TEMP(bTRIGGER := NOT BWTS_008, tDELAY := T#30S); // BWTS.ALARM_D
CC100_TEMP_HI := ALARM_D_CC_TEMP.ALARM;
ALARM_D_MCC_OFF(bTRIGGER := NOT TRUE, tDELAY := T#1S); // BWTS.ALARM_D
MCC_100_OFF := ALARM_D_MCC_OFF.ALARM;
ALARM_D_B117A_OFF(bTRIGGER := NOT TRUE, tDELAY := T#1S); // BWTS.ALARM_D
B_117A_OFF := ALARM_D_B117A_OFF.ALARM;
ALARM_D_B117B_OFF(bTRIGGER := NOT TRUE, tDELAY := T#1S); // BWTS.ALARM_D
B_117B_OFF := ALARM_D_B117B_OFF.ALARM;
ALARM_D_B117A_F(bTRIGGER := NOT TRUE, tDELAY := T#1S); // BWTS.ALARM_D
B_117A_F := ALARM_D_B117A_F.ALARM;
ALARM_D_B117B_F(bTRIGGER := NOT TRUE, tDELAY := T#1S); // BWTS.ALARM_D
B_117B_F := ALARM_D_B117B_F.ALARM;
ALARM_D_P171A_OFF(bTRIGGER := NOT TRUE, tDELAY := T#1S); // BWTS.ALARM_D
P_171A_OFF := ALARM_D_P171A_OFF.ALARM;
ALARM_D_P171B_OFF(bTRIGGER := NOT TRUE, tDELAY := T#1S); // BWTS.ALARM_D
P_171B_OFF := ALARM_D_P171B_OFF.ALARM;
ALARM_D_P171B_F(bTRIGGER := NOT TRUE, tDELAY := T#1S); // BWTS.ALARM_D
P_171B_F := ALARM_D_P171B_F.ALARM;
ALARM_D_P171A_F(bTRIGGER := NOT TRUE, tDELAY := T#1S); // BWTS.ALARM_D
P_171A_F := ALARM_D_P171A_F.ALARM;
ALARM_D_P232_TRIP(bTRIGGER := NOT TRUE, tDELAY := T#1S); // BWTS.ALARM_D
P_232_TRIP := ALARM_D_P232_TRIP.ALARM;
ALARM_D_P132_TRIP(bTRIGGER := NOT TRUE, tDELAY := T#1S); // BWTS.ALARM_D
P_132_TRIP := ALARM_D_P132_TRIP.ALARM;
ALARM_D_RF142A_E(bTRIGGER := NOT TRUE, tDELAY := T#1S); // BWTS.ALARM_D
RF_142A_E := ALARM_D_RF142A_E.ALARM;
ALARM_D_RF142B_E(bTRIGGER := NOT TRUE, tDELAY := T#1S); // BWTS.ALARM_D
RF_142B_E := ALARM_D_RF142B_E.ALARM;
ALARM_D_RF142C_E(bTRIGGER := NOT TRUE, tDELAY := T#1S); // BWTS.ALARM_D
RF_142C_E := ALARM_D_RF142C_E.ALARM;
(* (BST_S_01.COMPLETE OR BST_P_01.COMPLETE) AND B117A_SPD AND B117B_SPD; result not used *)
ALARM_D_BLR_SPD(bTRIGGER := _w1, tDELAY := T#15S); // BWTS.ALARM_D
BLR_BOTH_F := ALARM_D_BLR_SPD.ALARM;
(* (BST_S_06.COMPLETE OR BST_P_06.COMPLETE) AND P171A_SPD AND P171B_SPD; result not used *)
ALARM_D_SWP_SPD(bTRIGGER := _w2, tDELAY := T#15S); // BWTS.ALARM_D
SWFP_BOTH_F := ALARM_D_SWP_SPD.ALARM;
(* (BST_S_14.COMPLETE OR BST_P_14.COMPLETE) AND RFA_SPD AND RFB_SPD AND RFC_SPD; result not used *)
ALARM_D_RF_SPD(bTRIGGER := _w3, tDELAY := T#10S); // BWTS.ALARM_D
RF_ALL_SPD := ALARM_D_RF_SPD.ALARM;
ALARM_D_BLR_BYPASS(bTRIGGER := MF_B117_BP, tDELAY := T#1S); // BWTS.ALARM_D
BLR_BYPASS := ALARM_D_BLR_BYPASS.ALARM;
(* (BST_S_07.COMPLETE OR BST_P_07.COMPLETE) AND NOT LS_1111; result not used *)
ALARM_D_LS_1111(bTRIGGER := _w4, tDELAY := T#3S); // BWTS.ALARM_D
LS_1111_LL := ALARM_D_LS_1111.ALARM;
ALARM_D_LS_1141(bTRIGGER := NOT LS_1141, tDELAY := T#30S); // BWTS.ALARM_D
LS_1141_HI := ALARM_D_LS_1141.ALARM;
(* NOT RFA_DISABLE AND NOT ZS_1112A_OPD; result not used *)
ALARM_D_ZS_1112A_CL(bTRIGGER := _w5, tDELAY := T#1S); // BWTS.ALARM_D
ZS_1112A_CL := ALARM_D_ZS_1112A_CL.ALARM;
(* NOT RFB_DISABLE AND NOT ZS_1113A_OPD; result not used *)
ALARM_D_ZS_1113A_CL(bTRIGGER := _w6, tDELAY := T#1S); // BWTS.ALARM_D
ZS_1113A_CL := ALARM_D_ZS_1113A_CL.ALARM;
(* NOT RFC_DISABLE AND NOT ZS_1114A_OPD; result not used *)
ALARM_D_ZS_1114A_CL(bTRIGGER := _w7, tDELAY := T#1S); // BWTS.ALARM_D
ZS_1114A_CL := ALARM_D_ZS_1114A_CL.ALARM;
(* RFA_DISABLE AND ZS_1112A_OPD; result not used *)
ALARM_D_ZS_1112A_OP(bTRIGGER := _w8, tDELAY := T#1S); // BWTS.ALARM_D
ZS_1112A_OP := ALARM_D_ZS_1112A_OP.ALARM;
(* RFB_DISABLE AND ZS_1113A_OPD; result not used *)
ALARM_D_ZS_1113A_OP(bTRIGGER := _w9, tDELAY := T#1S); // BWTS.ALARM_D
ZS_1113A_OP := ALARM_D_ZS_1113A_OP.ALARM;
(* RFC_DISABLE AND ZS_1114A_OPD; result not used *)
ALARM_D_ZS_1114A_OP(bTRIGGER := _w10, tDELAY := T#1S); // BWTS.ALARM_D
ZS_1114A_OP := ALARM_D_ZS_1114A_OP.ALARM;
(* NOT (BAL_IN_STBD OR DEBAL_IN_STBD) AND WBP01_RUN; result not used *)
ALARM_D_WBP_01_AL(bTRIGGER := _w11, tDELAY := T#1S); // BWTS.ALARM_D
WBP_01_AL := ALARM_D_WBP_01_AL.ALARM;
(* NOT (BAL_IN_PORT OR DEBAL_IN_PORT) AND WBP02_RUN; result not used *)
ALARM_D_WBP_02_AL(bTRIGGER := _w12, tDELAY := T#1S); // BWTS.ALARM_D
WBP_02_AL := ALARM_D_WBP_02_AL.ALARM;
(* (BST_S_08.COMPLETE OR DST_S_04.COMPLETE) AND WBP01_SPD; result not used *)
ALARM_D_WBP_01_FAULT(bTRIGGER := _w13, tDELAY := T#1S); // BWTS.ALARM_D
WBP_01_FAULT := ALARM_D_WBP_01_FAULT.ALARM;
(* (BST_P_08.COMPLETE OR DST_P_04.COMPLETE) AND WBP02_SPD; result not used *)
ALARM_D_WBP_02_FAULT(bTRIGGER := _w14, tDELAY := T#1S); // BWTS.ALARM_D
WBP_02_FAULT := ALARM_D_WBP_02_FAULT.ALARM;
(* NOT STR_IN_STBD AND GSP01_RUN AND NOT TRUE; result not used *)
ALARM_D_GSP_01_AL(bTRIGGER := _w15, tDELAY := T#1S); // BWTS.ALARM_D
GSP_01_AL := ALARM_D_GSP_01_AL.ALARM;
(* NOT STR_IN_STBD AND GSP02_RUN AND NOT TRUE; result not used *)
ALARM_D_GSP_02_AL(bTRIGGER := _w16, tDELAY := T#1S); // BWTS.ALARM_D
GSP_02_AL := ALARM_D_GSP_02_AL.ALARM;
(* SST_S_02.COMPLETE AND GSP01_SEL AND GSP01_SPD; result not used *)
ALARM_D_GSP_01_FAULT(bTRIGGER := _w17, tDELAY := T#1S); // BWTS.ALARM_D
GSP_01_FAULT := ALARM_D_GSP_01_FAULT.ALARM;
(* SST_S_02.COMPLETE AND GSP02_SEL AND GSP02_SPD; result not used *)
ALARM_D_GSP_02_FAULT(bTRIGGER := _w18, tDELAY := T#1S); // BWTS.ALARM_D
GSP_02_FAULT := ALARM_D_GSP_02_FAULT.ALARM;
(* SEL(NU_CROSS, SEQ_DEBAL_ST_S.TON_0.Q AND NOT TRUE, NOT TRUE AND SEQ_DEBAL_ST_P.TON_0.Q); result not used *)
ALARM_D_DPS_1321(bTRIGGER := _w19, tDELAY := T#1S); // BWTS.ALARM_D
DPS_1321 := ALARM_D_DPS_1321.ALARM;
(* SEL(NU_CROSS, SEQ_DEBAL_ST_P.TON_0.Q AND NOT TRUE, NOT TRUE AND SEQ_DEBAL_ST_S.TON_0.Q); result not used *)
ALARM_D_DPS_2321(bTRIGGER := _w20, tDELAY := T#1S); // BWTS.ALARM_D
DPS_2321 := ALARM_D_DPS_2321.ALARM;
ALARM_D_RFS_1131(bTRIGGER := NOT TRUE AND BST_S_13.COMPLETE, tDELAY := T#1S); // BWTS.ALARM_D
RFS_1131 := ALARM_D_RFS_1131.ALARM;
ALARM_D_RFS_2131(bTRIGGER := NOT TRUE AND BST_P_13.COMPLETE, tDELAY := T#1S); // BWTS.ALARM_D
RFS_2131 := ALARM_D_RFS_2131.ALARM;
TON_AIT151_E(IN := AIT_151_ST, PT := MS_TRO_STABLE); // TON
ALARM_D_AIT_151_E(bTRIGGER := TON_AIT151_E.Q AND FALSE, tDELAY := T#300S); // BWTS.ALARM_D
AIT_151_E := ALARM_D_AIT_151_E.ALARM;
TON_AIT151_F(IN := AIT_151_ST, PT := MS_TRO_STABLE); // TON
ALARM_D_AIT_151_F(bTRIGGER := TON_AIT151_F.Q AND FALSE, tDELAY := T#600S); // BWTS.ALARM_D
AIT_151_F := ALARM_D_AIT_151_F.ALARM;
TON_AIT251_E(IN := AIT_251_ST, PT := MS_TRO_STABLE); // TON
ALARM_D_AIT_251_E(bTRIGGER := TON_AIT251_E.Q AND FALSE, tDELAY := T#300S); // BWTS.ALARM_D
AIT_251_E := ALARM_D_AIT_251_E.ALARM;
TON_AIT251_F(IN := AIT_251_ST, PT := MS_TRO_STABLE); // TON
ALARM_D_AIT_251_F(bTRIGGER := TON_AIT251_F.Q AND FALSE, tDELAY := T#600S); // BWTS.ALARM_D
AIT_251_F := ALARM_D_AIT_251_F.ALARM;
ALARM_D_GAS_LEAK_AL(bTRIGGER := NOT TRUE, tDELAY := T#3S); // BWTS.ALARM_D
GAS_LEAK_AL := ALARM_D_GAS_LEAK_AL.ALARM;
ALARM_D_LS_1901_HH(bTRIGGER := LS_1901_HI, tDELAY := T#30S); // BWTS.ALARM_D
LS_1901_HH := ALARM_D_LS_1901_HH.ALARM;

END_PROGRAM

// Device/Application/Logic/0.ALARM/ALARM_INTERLOCK_D_2
PROGRAM ALARM_INTERLOCK_D_2
VAR
	ALARM_D_SYS_BYPASS_1,
	ALARM_D_SYS_BYPASS_2,
	ALARM_D_SYS_BYPASS_3,
	ALARM_D_SYS_BYPASS_4,
	ALARM_D_BAL_VV_AL_S,
	ALARM_D_BAL_VV_AL_P,
	
	ALARM_D_DEBAL_VV_AL_S,
	ALARM_D_DEBAL_VV_AL_P,
	
	ALARM_D_STR_VV_AL_S,
	ALARM_D_RH_ELECT,
	ALARM_D_RH_AIT1121,
	ALARM_D_RH_AIT1122,
	ALARM_D_RH_AIT1123,
	ALARM_D_RH_P171A,
	ALARM_D_RH_P171B,
	ALARM_D_RH_P132,
	ALARM_D_RH_P232,
	
	
	ALARM_D_RH_AIT151,
	ALARM_D_RH_AIT251,
	
	ALARM_D_PR_FAN,
	ALARM_D_BR_FAN
	: BWTS.ALARM_D;
END_VAR
VAR // added by the converter: edge detectors and wires of the graphical bodies
    _w1, _w2, _w3, _w4, _w5, _w6, _w7, _w8, _w9, _w10, _w11, _w12, _w13, _w14, _w15, _w16, _w17, _w18, _w19, _w20, _w21 : ANY;
END_VAR

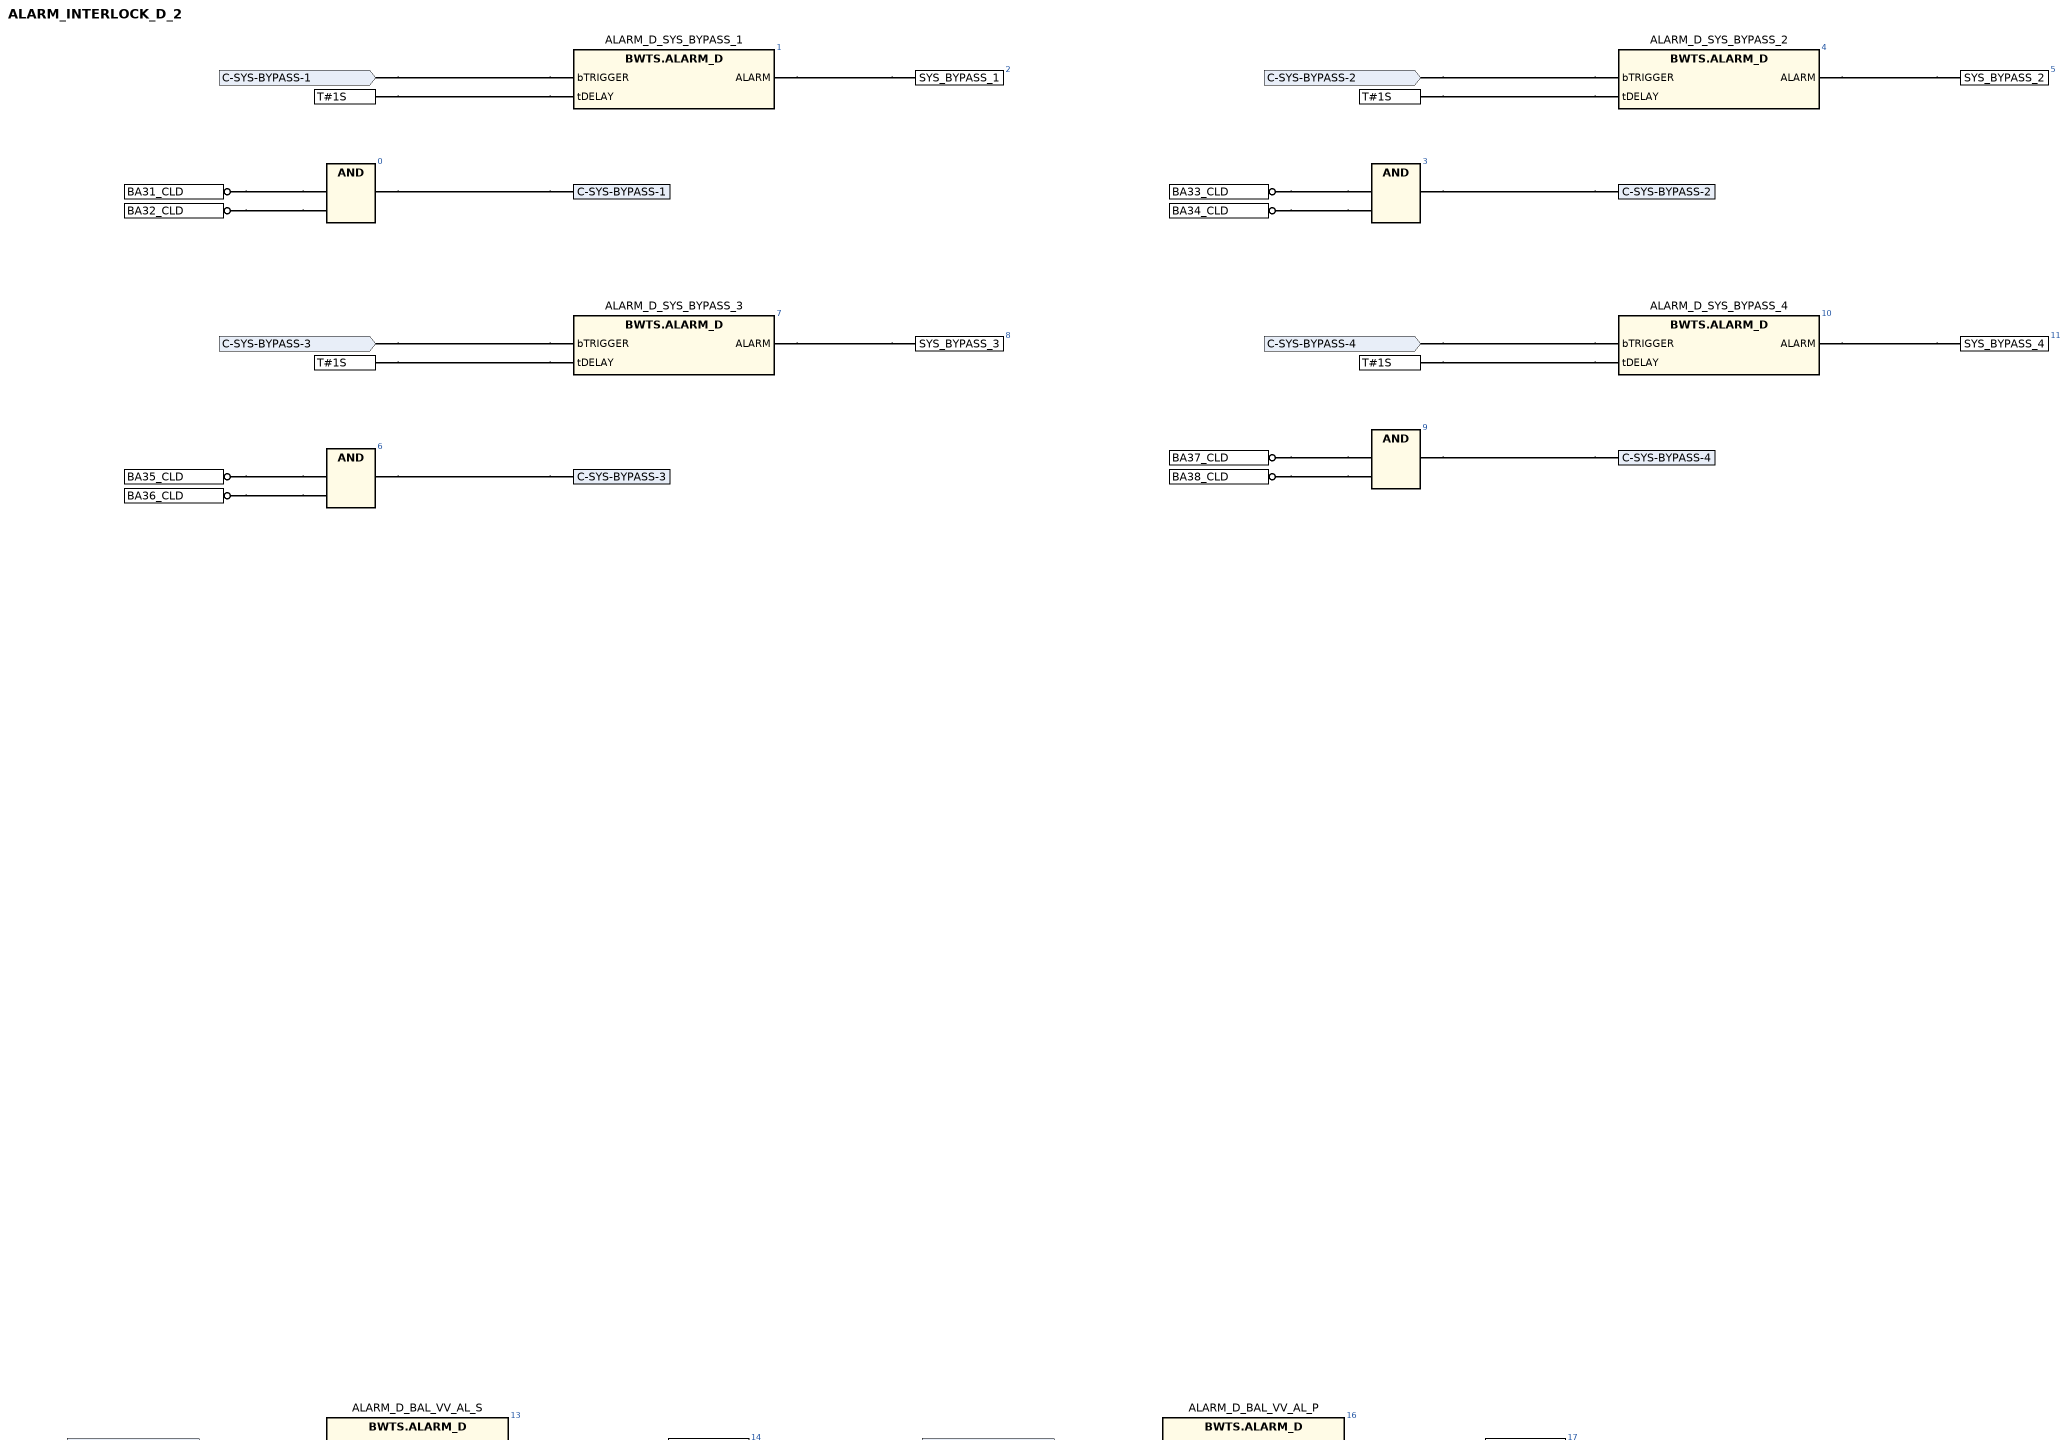
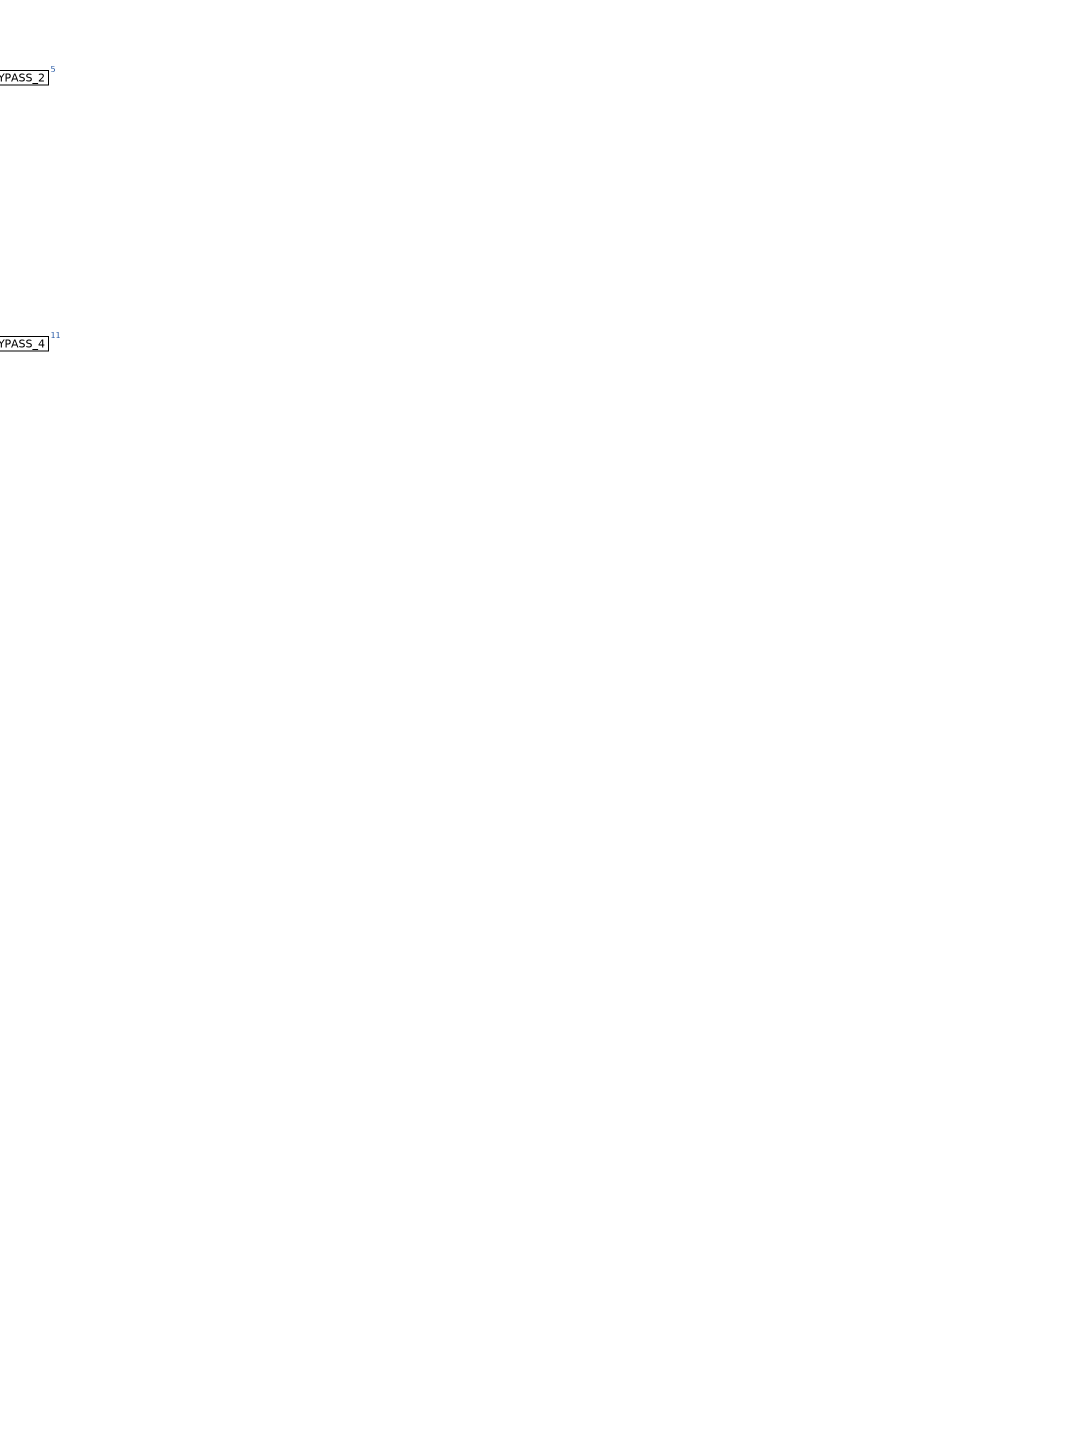
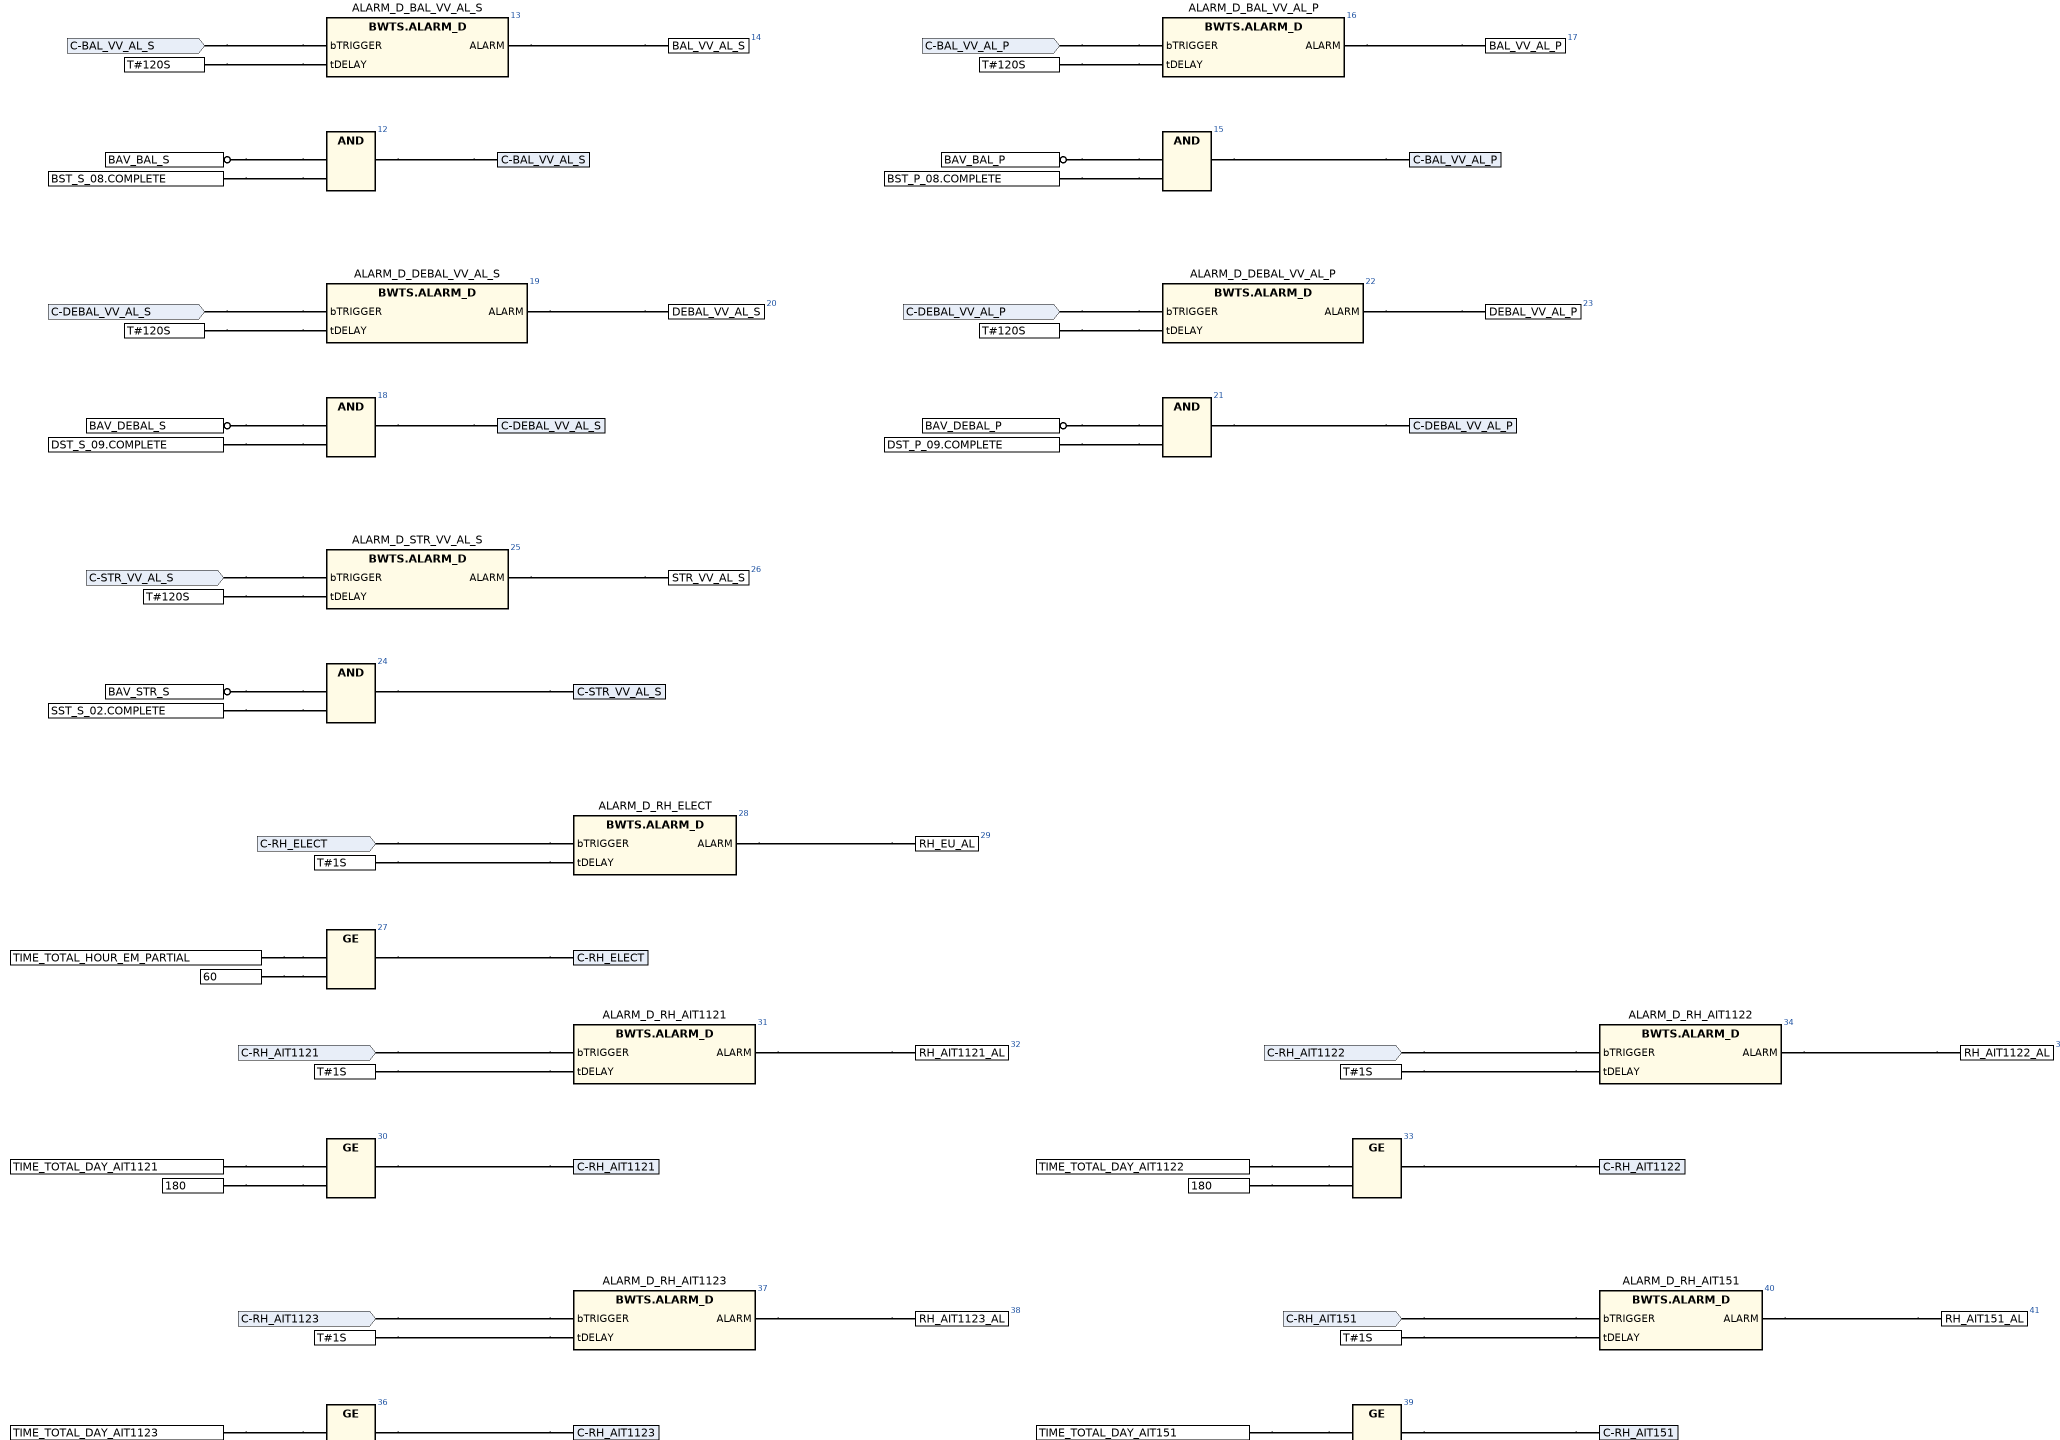
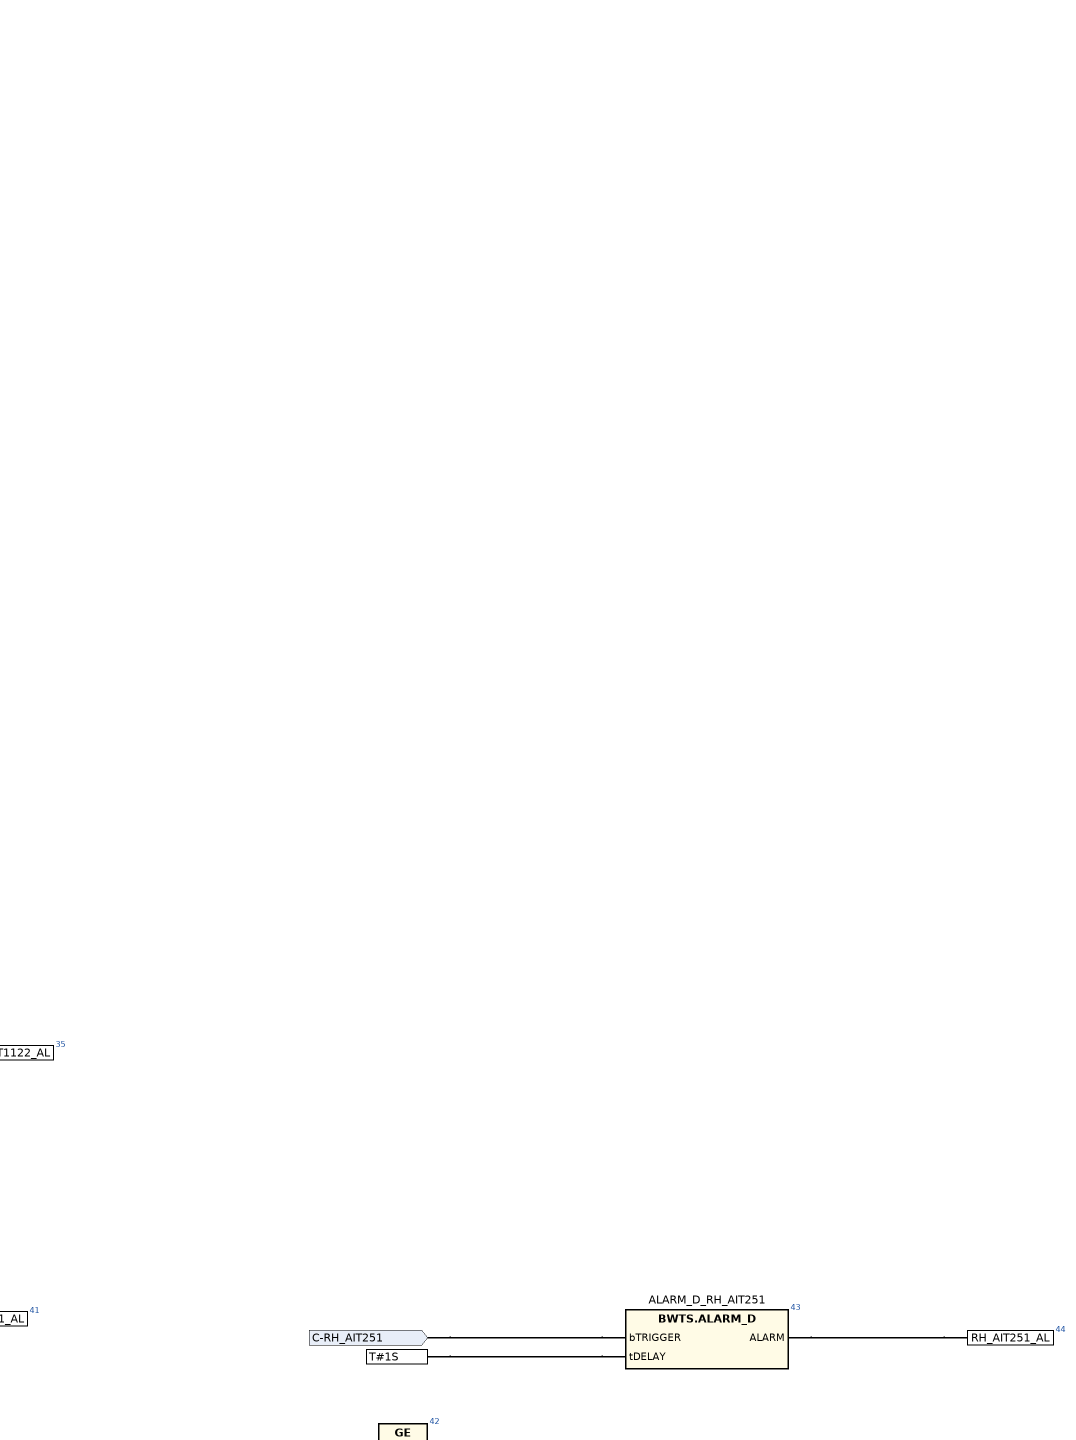
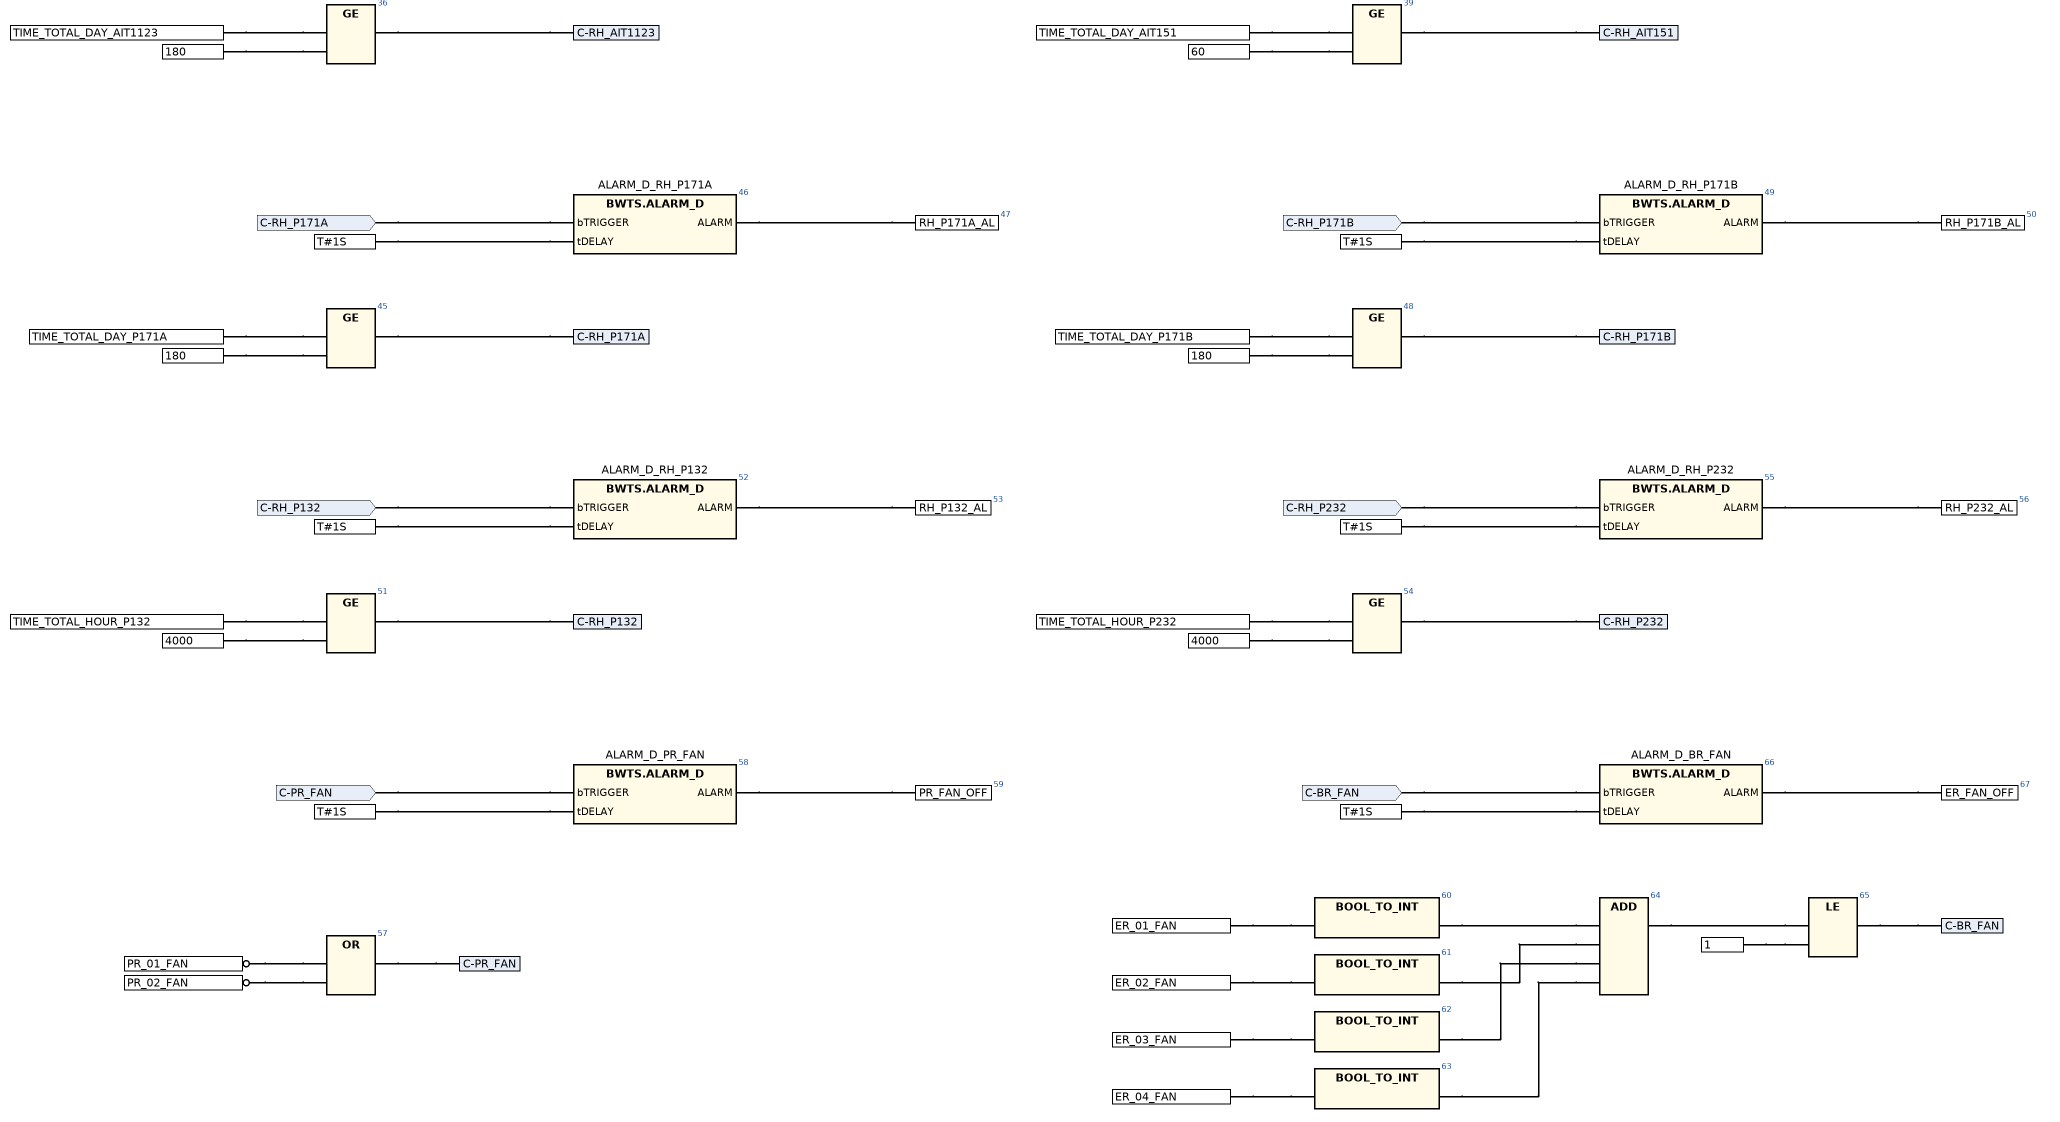
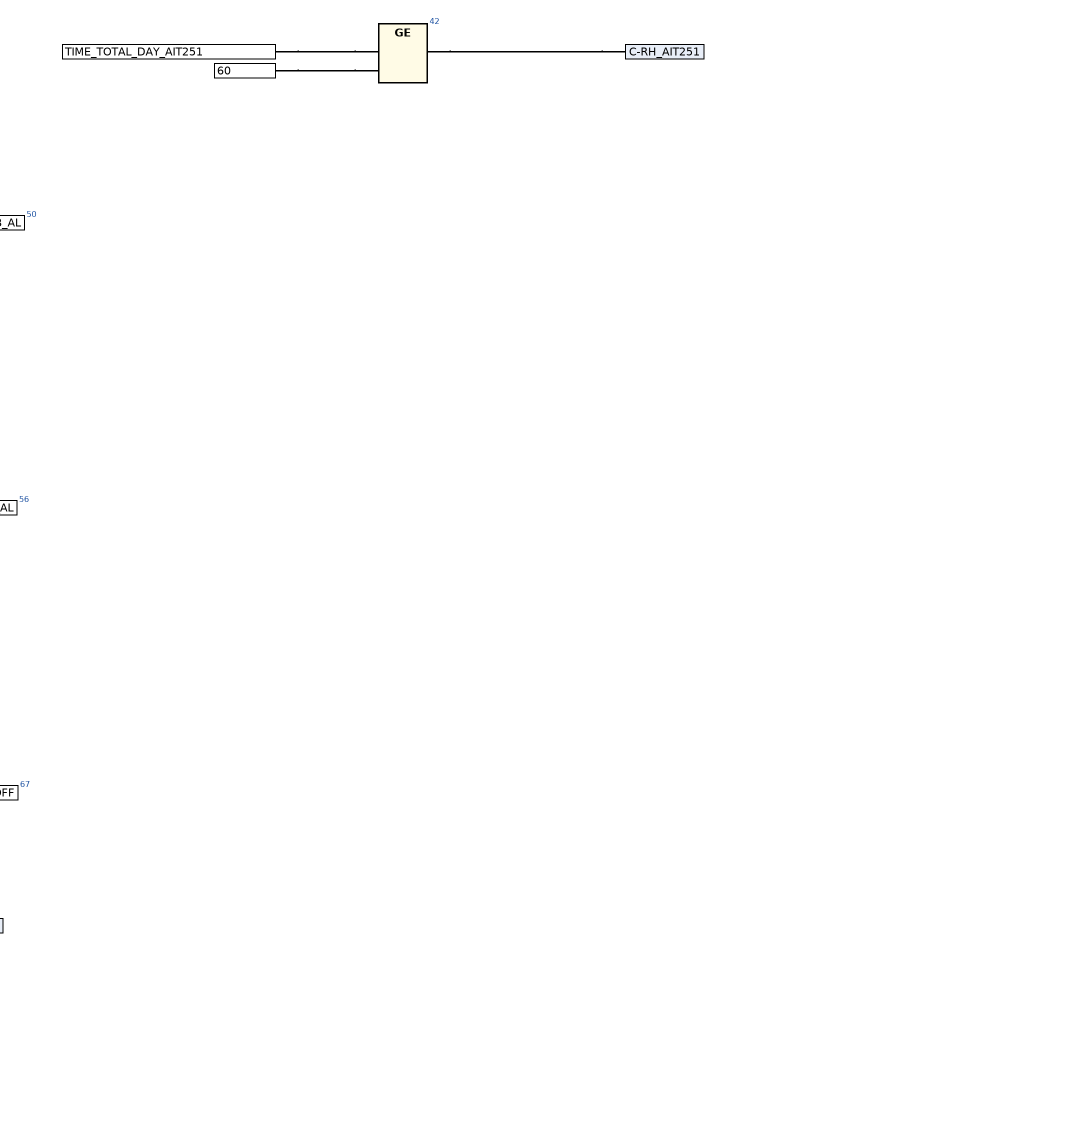
(* NOT BA31_CLD AND NOT BA32_CLD; result not used *)
ALARM_D_SYS_BYPASS_1(bTRIGGER := _w1, tDELAY := T#1S); // BWTS.ALARM_D
SYS_BYPASS_1 := ALARM_D_SYS_BYPASS_1.ALARM;
(* NOT BA33_CLD AND NOT BA34_CLD; result not used *)
ALARM_D_SYS_BYPASS_2(bTRIGGER := _w2, tDELAY := T#1S); // BWTS.ALARM_D
SYS_BYPASS_2 := ALARM_D_SYS_BYPASS_2.ALARM;
(* NOT BA35_CLD AND NOT BA36_CLD; result not used *)
ALARM_D_SYS_BYPASS_3(bTRIGGER := _w3, tDELAY := T#1S); // BWTS.ALARM_D
SYS_BYPASS_3 := ALARM_D_SYS_BYPASS_3.ALARM;
(* NOT BA37_CLD AND NOT BA38_CLD; result not used *)
ALARM_D_SYS_BYPASS_4(bTRIGGER := _w4, tDELAY := T#1S); // BWTS.ALARM_D
SYS_BYPASS_4 := ALARM_D_SYS_BYPASS_4.ALARM;
(* NOT BAV_BAL_S AND BST_S_08.COMPLETE; result not used *)
ALARM_D_BAL_VV_AL_S(bTRIGGER := _w5, tDELAY := T#120S); // BWTS.ALARM_D
BAL_VV_AL_S := ALARM_D_BAL_VV_AL_S.ALARM;
(* NOT BAV_BAL_P AND BST_P_08.COMPLETE; result not used *)
ALARM_D_BAL_VV_AL_P(bTRIGGER := _w6, tDELAY := T#120S); // BWTS.ALARM_D
BAL_VV_AL_P := ALARM_D_BAL_VV_AL_P.ALARM;
(* NOT BAV_DEBAL_S AND DST_S_09.COMPLETE; result not used *)
ALARM_D_DEBAL_VV_AL_S(bTRIGGER := _w7, tDELAY := T#120S); // BWTS.ALARM_D
DEBAL_VV_AL_S := ALARM_D_DEBAL_VV_AL_S.ALARM;
(* NOT BAV_DEBAL_P AND DST_P_09.COMPLETE; result not used *)
ALARM_D_DEBAL_VV_AL_P(bTRIGGER := _w8, tDELAY := T#120S); // BWTS.ALARM_D
DEBAL_VV_AL_P := ALARM_D_DEBAL_VV_AL_P.ALARM;
(* NOT BAV_STR_S AND SST_S_02.COMPLETE; result not used *)
ALARM_D_STR_VV_AL_S(bTRIGGER := _w9, tDELAY := T#120S); // BWTS.ALARM_D
STR_VV_AL_S := ALARM_D_STR_VV_AL_S.ALARM;
(* TIME_TOTAL_HOUR_EM_PARTIAL >= 60; result not used *)
ALARM_D_RH_ELECT(bTRIGGER := _w10, tDELAY := T#1S); // BWTS.ALARM_D
RH_EU_AL := ALARM_D_RH_ELECT.ALARM;
(* TIME_TOTAL_DAY_AIT1121 >= 180; result not used *)
ALARM_D_RH_AIT1121(bTRIGGER := _w11, tDELAY := T#1S); // BWTS.ALARM_D
RH_AIT1121_AL := ALARM_D_RH_AIT1121.ALARM;
(* TIME_TOTAL_DAY_AIT1122 >= 180; result not used *)
ALARM_D_RH_AIT1122(bTRIGGER := _w12, tDELAY := T#1S); // BWTS.ALARM_D
RH_AIT1122_AL := ALARM_D_RH_AIT1122.ALARM;
(* TIME_TOTAL_DAY_AIT1123 >= 180; result not used *)
ALARM_D_RH_AIT1123(bTRIGGER := _w13, tDELAY := T#1S); // BWTS.ALARM_D
RH_AIT1123_AL := ALARM_D_RH_AIT1123.ALARM;
(* TIME_TOTAL_DAY_AIT151 >= 60; result not used *)
ALARM_D_RH_AIT151(bTRIGGER := _w14, tDELAY := T#1S); // BWTS.ALARM_D
RH_AIT151_AL := ALARM_D_RH_AIT151.ALARM;
(* TIME_TOTAL_DAY_AIT251 >= 60; result not used *)
ALARM_D_RH_AIT251(bTRIGGER := _w15, tDELAY := T#1S); // BWTS.ALARM_D
RH_AIT251_AL := ALARM_D_RH_AIT251.ALARM;
(* TIME_TOTAL_DAY_P171A >= 180; result not used *)
ALARM_D_RH_P171A(bTRIGGER := _w16, tDELAY := T#1S); // BWTS.ALARM_D
RH_P171A_AL := ALARM_D_RH_P171A.ALARM;
(* TIME_TOTAL_DAY_P171B >= 180; result not used *)
ALARM_D_RH_P171B(bTRIGGER := _w17, tDELAY := T#1S); // BWTS.ALARM_D
RH_P171B_AL := ALARM_D_RH_P171B.ALARM;
(* TIME_TOTAL_HOUR_P132 >= 4000; result not used *)
ALARM_D_RH_P132(bTRIGGER := _w18, tDELAY := T#1S); // BWTS.ALARM_D
RH_P132_AL := ALARM_D_RH_P132.ALARM;
(* TIME_TOTAL_HOUR_P232 >= 4000; result not used *)
ALARM_D_RH_P232(bTRIGGER := _w19, tDELAY := T#1S); // BWTS.ALARM_D
RH_P232_AL := ALARM_D_RH_P232.ALARM;
(* NOT PR_01_FAN OR NOT PR_02_FAN; result not used *)
ALARM_D_PR_FAN(bTRIGGER := _w20, tDELAY := T#1S); // BWTS.ALARM_D
PR_FAN_OFF := ALARM_D_PR_FAN.ALARM;
(* BOOL_TO_INT(ER_01_FAN) + BOOL_TO_INT(ER_02_FAN) + BOOL_TO_INT(ER_03_FAN) + BOOL_TO_INT(ER_04_FAN) <= 1; result not used *)
ALARM_D_BR_FAN(bTRIGGER := _w21, tDELAY := T#1S); // BWTS.ALARM_D
ER_FAN_OFF := ALARM_D_BR_FAN.ALARM;

END_PROGRAM

// Device/Application/Logic/0.ALARM/ALARM_RECTIFIER
PROGRAM ALARM_RECTIFIER
VAR
	ALARM_A_REC1017 : BWTS.ALARM_A;
	ALARM_A_REC1018 : BWTS.ALARM_A;
	ALARM_A_REC1019 : BWTS.ALARM_A;
	ALARM_A_REC1020 : BWTS.ALARM_A;
	ALARM_A_REC1021 : BWTS.ALARM_A;
	ALARM_A_REC1027 : BWTS.ALARM_A;
          
 	ALARM_A_REC2017 : BWTS.ALARM_A;
	ALARM_A_REC2018 : BWTS.ALARM_A;
	ALARM_A_REC2019 : BWTS.ALARM_A;
	ALARM_A_REC2020 : BWTS.ALARM_A;
	ALARM_A_REC2021 : BWTS.ALARM_A;
	ALARM_A_REC2027 : BWTS.ALARM_A;
	
	ALARM_A_REC3017 : BWTS.ALARM_A;
	ALARM_A_REC3018 : BWTS.ALARM_A;
	ALARM_A_REC3019 : BWTS.ALARM_A;
	ALARM_A_REC3020 : BWTS.ALARM_A;
	ALARM_A_REC3021 : BWTS.ALARM_A;
	ALARM_A_REC3027 : BWTS.ALARM_A;
END_VAR


ALARM_A_REC1017(bTRIGGER := TRUE, rVALUE := REC1017, rLIMIT_HH := MS_100D_A_HH , rLIMIT_HI := MS_100D_A_HI, tDELAY_HH := TD_100D_A_HH,  tDELAY_HI := TD_100D_A_HI, HH => REC1017_HH, HI => REC1017_HI );
ALARM_A_REC1018(bTRIGGER := TRUE, rVALUE := REC1018, rLIMIT_HH := MS_100D_V_HH , rLIMIT_HI := MS_100D_V_HI, tDELAY_HH := TD_100D_V_HH,  tDELAY_HI := TD_100D_V_HI, HH => REC1018_HH, HI => REC1018_HI );
ALARM_A_REC1019(bTRIGGER := TRUE, rVALUE := REC1019, rLIMIT_HH := MS_MD_TEMP_HH , rLIMIT_HI := MS_MD_TEMP_HI, tDELAY_HH := TD_MD_TEMP_HH,  tDELAY_HI := TD_MD_TEMP_HI, HH => REC1019_HH, HI => REC1019_HI );
ALARM_A_REC1020(bTRIGGER := TRUE, rVALUE := REC1020, rLIMIT_HH := MS_MD_TEMP_HH , rLIMIT_HI := MS_MD_TEMP_HI, tDELAY_HH := TD_MD_TEMP_HH,  tDELAY_HI := TD_MD_TEMP_HI, HH => REC1020_HH, HI => REC1020_HI );
ALARM_A_REC1021(bTRIGGER := TRUE, rVALUE := REC1021, rLIMIT_HH := MS_MD_TEMP_HH , rLIMIT_HI := MS_MD_TEMP_HI, tDELAY_HH := TD_MD_TEMP_HH,  tDELAY_HI := TD_MD_TEMP_HI, HH => REC1021_HH, HI => REC1021_HI );
ALARM_A_REC1027(bTRIGGER := TRUE, rVALUE := REC1027, rLIMIT_HH := MS_RF_TEMP_HH , rLIMIT_HI := MS_RF_TEMP_HI, tDELAY_HH := TD_RF_TEMP_HH,  tDELAY_HI := TD_RF_TEMP_HI, HH => REC1027_HH, HI => REC1027_HI );

ALARM_A_REC2017(bTRIGGER := TRUE, rVALUE := REC2017, rLIMIT_HH := MS_100D_A_HH, rLIMIT_HI := MS_100D_A_HI, tDELAY_HH := TD_100D_A_HH,  tDELAY_HI := TD_100D_A_HI, HH => REC2017_HH, HI => REC2017_HI );
ALARM_A_REC2018(bTRIGGER := TRUE, rVALUE := REC2018, rLIMIT_HH := MS_100D_V_HH, rLIMIT_HI := MS_100D_V_HI, tDELAY_HH := TD_100D_V_HH,  tDELAY_HI := TD_100D_V_HI, HH => REC2018_HH, HI => REC2018_HI );
ALARM_A_REC2019(bTRIGGER := TRUE, rVALUE := REC2019, rLIMIT_HH := MS_MD_TEMP_HH , rLIMIT_HI := MS_MD_TEMP_HI, tDELAY_HH := TD_MD_TEMP_HH,  tDELAY_HI := TD_MD_TEMP_HI, HH => REC2019_HH, HI => REC2019_HI );
ALARM_A_REC2020(bTRIGGER := TRUE, rVALUE := REC2020, rLIMIT_HH := MS_MD_TEMP_HH , rLIMIT_HI := MS_MD_TEMP_HI, tDELAY_HH := TD_MD_TEMP_HH,  tDELAY_HI := TD_MD_TEMP_HI, HH => REC2020_HH, HI => REC2020_HI );
ALARM_A_REC2021(bTRIGGER := TRUE, rVALUE := REC2021, rLIMIT_HH := MS_MD_TEMP_HH , rLIMIT_HI := MS_MD_TEMP_HI, tDELAY_HH := TD_MD_TEMP_HH,  tDELAY_HI := TD_MD_TEMP_HI, HH => REC2021_HH, HI => REC2021_HI );
ALARM_A_REC2027(bTRIGGER := TRUE, rVALUE := REC2027, rLIMIT_HH := MS_RF_TEMP_HH , rLIMIT_HI := MS_RF_TEMP_HI, tDELAY_HH := TD_RF_TEMP_HH,  tDELAY_HI := TD_RF_TEMP_HI, HH => REC2027_HH, HI => REC2027_HI );

ALARM_A_REC3017(bTRIGGER := TRUE, rVALUE := REC3017, rLIMIT_HH := MS_100D_A_HH, rLIMIT_HI := MS_100D_A_HI, tDELAY_HH := TD_100D_A_HH,  tDELAY_HI := TD_100D_A_HI, HH => REC3017_HH, HI => REC3017_HI );
ALARM_A_REC3018(bTRIGGER := TRUE, rVALUE := REC3018, rLIMIT_HH := MS_100D_V_HH, rLIMIT_HI := MS_100D_V_HI, tDELAY_HH := TD_100D_V_HH,  tDELAY_HI := TD_100D_V_HI, HH => REC3018_HH, HI => REC3018_HI );
ALARM_A_REC3019(bTRIGGER := TRUE, rVALUE := REC3019, rLIMIT_HH := MS_MD_TEMP_HH , rLIMIT_HI := MS_MD_TEMP_HI, tDELAY_HH := TD_MD_TEMP_HH,  tDELAY_HI := TD_MD_TEMP_HI, HH => REC3019_HH, HI => REC3019_HI );
ALARM_A_REC3020(bTRIGGER := TRUE, rVALUE := REC3020, rLIMIT_HH := MS_MD_TEMP_HH , rLIMIT_HI := MS_MD_TEMP_HI, tDELAY_HH := TD_MD_TEMP_HH,  tDELAY_HI := TD_MD_TEMP_HI, HH => REC3020_HH, HI => REC3020_HI );
ALARM_A_REC3021(bTRIGGER := TRUE, rVALUE := REC3021, rLIMIT_HH := MS_MD_TEMP_HH , rLIMIT_HI := MS_MD_TEMP_HI, tDELAY_HH := TD_MD_TEMP_HH,  tDELAY_HI := TD_MD_TEMP_HI, HH => REC3021_HH, HI => REC3021_HI );
ALARM_A_REC3027(bTRIGGER := TRUE, rVALUE := REC3027, rLIMIT_HH := MS_RF_TEMP_HH , rLIMIT_HI := MS_RF_TEMP_HI, tDELAY_HH := TD_RF_TEMP_HH,  tDELAY_HI := TD_RF_TEMP_HI, HH => REC3027_HH, HI => REC3027_HI );

END_PROGRAM

// Device/Application/Logic/0.ALARM/ALARM_TRO
PROGRAM ALARM_TRO
VAR
	ALARM_TRO_BAL_S: BWTS.ALARM_TRO;
	ALARM_TRO_BAL_P: BWTS.ALARM_TRO;
	
	ALARM_TRO_DEBAL_S: BWTS.ALARM_TRO;
	ALARM_TRO_DEBAL_P: BWTS.ALARM_TRO;
	
	ALARM_TRO_STR: BWTS.ALARM_TRO;	
END_VAR
VAR // added by the converter: edge detectors and wires of the graphical bodies
    _w1, _w2, _w3, _w4, _w5, _w6, _w7, _w8, _w9, _w10 : ANY;
END_VAR

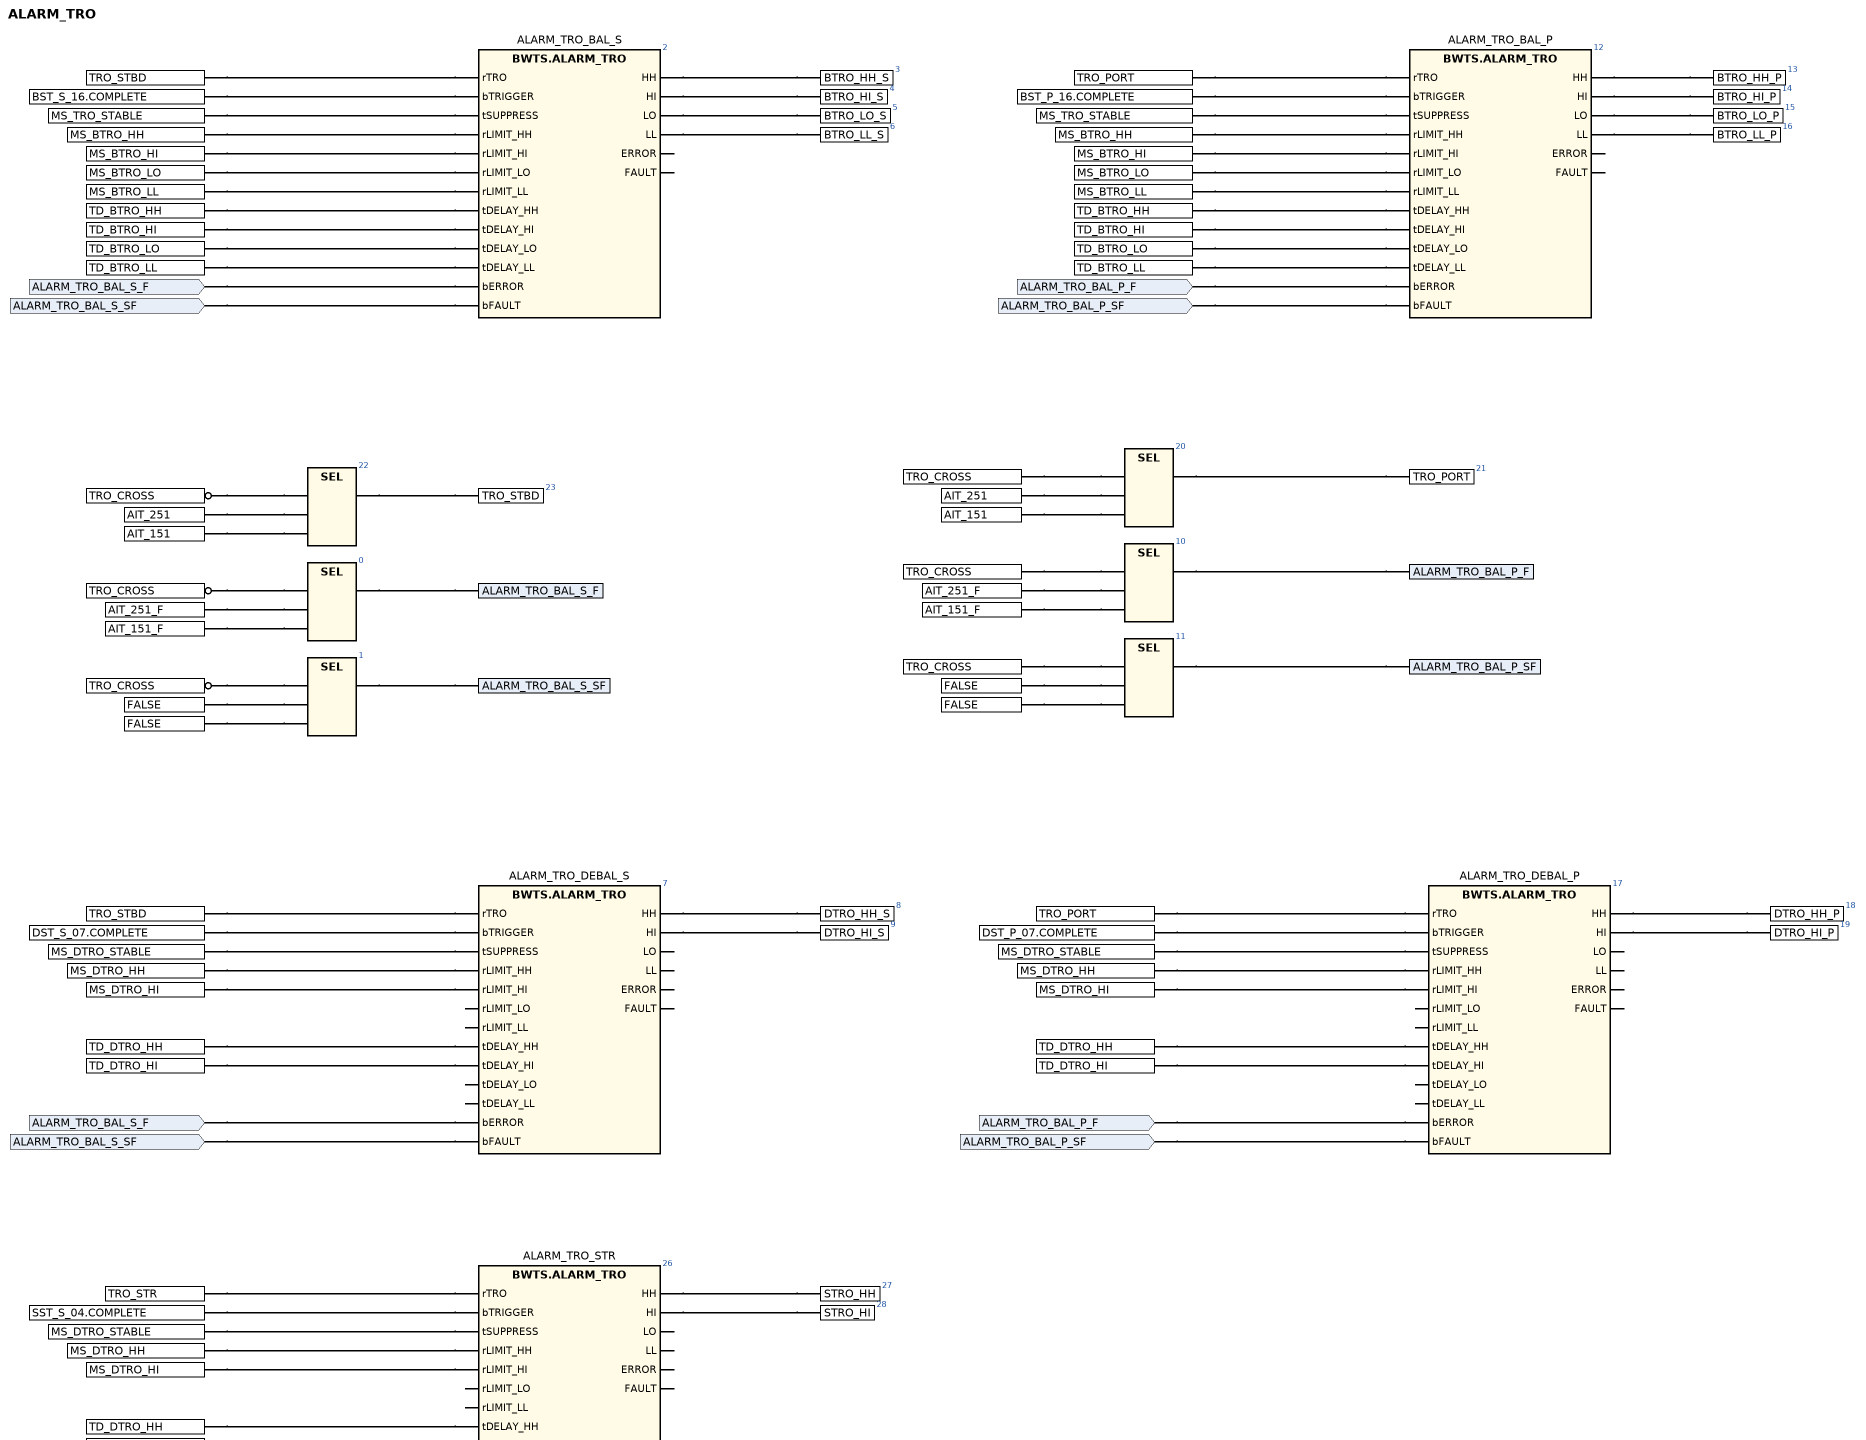
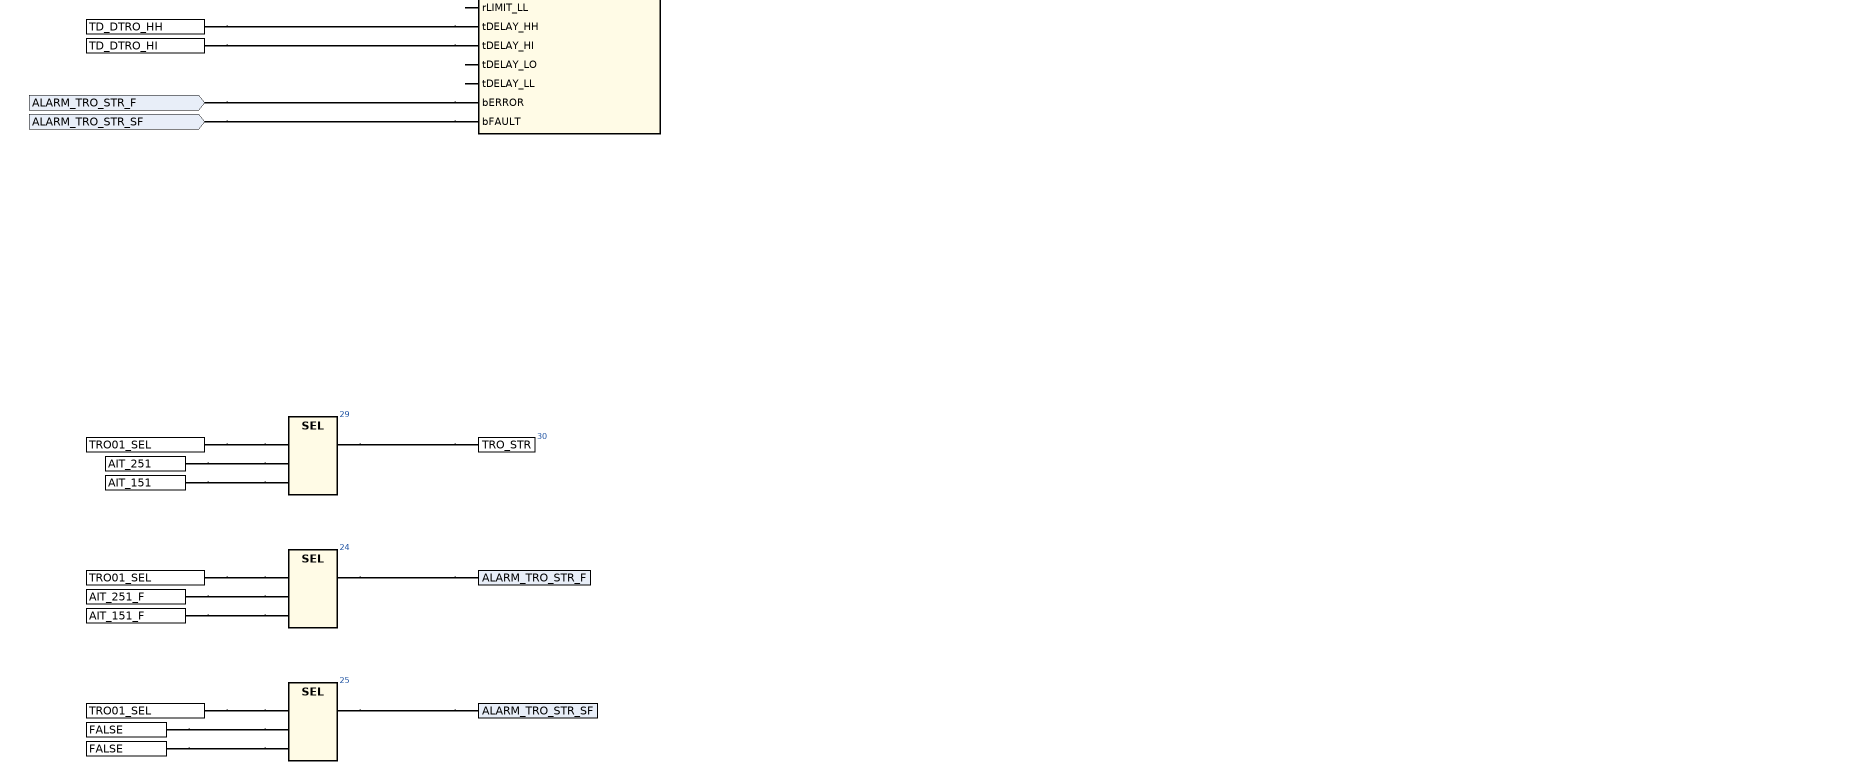
(* SEL(NOT TRO_CROSS, AIT_251_F, AIT_151_F); result not used *)
(* SEL(NOT TRO_CROSS, FALSE, FALSE); result not used *)
ALARM_TRO_BAL_S(
    rTRO := TRO_STBD,
    bTRIGGER := BST_S_16.COMPLETE,
    tSUPPRESS := MS_TRO_STABLE,
    rLIMIT_HH := MS_BTRO_HH,
    rLIMIT_HI := MS_BTRO_HI,
    rLIMIT_LO := MS_BTRO_LO,
    rLIMIT_LL := MS_BTRO_LL,
    tDELAY_HH := TD_BTRO_HH,
    tDELAY_HI := TD_BTRO_HI,
    tDELAY_LO := TD_BTRO_LO,
    tDELAY_LL := TD_BTRO_LL,
    bERROR := _w1,
    bFAULT := _w2); // BWTS.ALARM_TRO
BTRO_HH_S := ALARM_TRO_BAL_S.HH;
BTRO_HI_S := ALARM_TRO_BAL_S.HI;
BTRO_LO_S := ALARM_TRO_BAL_S.LO;
BTRO_LL_S := ALARM_TRO_BAL_S.LL;
ALARM_TRO_DEBAL_S(
    rTRO := TRO_STBD,
    bTRIGGER := DST_S_07.COMPLETE,
    tSUPPRESS := MS_DTRO_STABLE,
    rLIMIT_HH := MS_DTRO_HH,
    rLIMIT_HI := MS_DTRO_HI,
    tDELAY_HH := TD_DTRO_HH,
    tDELAY_HI := TD_DTRO_HI,
    bERROR := _w3,
    bFAULT := _w4); // BWTS.ALARM_TRO
DTRO_HH_S := ALARM_TRO_DEBAL_S.HH;
DTRO_HI_S := ALARM_TRO_DEBAL_S.HI;
(* SEL(TRO_CROSS, AIT_251_F, AIT_151_F); result not used *)
(* SEL(TRO_CROSS, FALSE, FALSE); result not used *)
ALARM_TRO_BAL_P(
    rTRO := TRO_PORT,
    bTRIGGER := BST_P_16.COMPLETE,
    tSUPPRESS := MS_TRO_STABLE,
    rLIMIT_HH := MS_BTRO_HH,
    rLIMIT_HI := MS_BTRO_HI,
    rLIMIT_LO := MS_BTRO_LO,
    rLIMIT_LL := MS_BTRO_LL,
    tDELAY_HH := TD_BTRO_HH,
    tDELAY_HI := TD_BTRO_HI,
    tDELAY_LO := TD_BTRO_LO,
    tDELAY_LL := TD_BTRO_LL,
    bERROR := _w5,
    bFAULT := _w6); // BWTS.ALARM_TRO
BTRO_HH_P := ALARM_TRO_BAL_P.HH;
BTRO_HI_P := ALARM_TRO_BAL_P.HI;
BTRO_LO_P := ALARM_TRO_BAL_P.LO;
BTRO_LL_P := ALARM_TRO_BAL_P.LL;
ALARM_TRO_DEBAL_P(
    rTRO := TRO_PORT,
    bTRIGGER := DST_P_07.COMPLETE,
    tSUPPRESS := MS_DTRO_STABLE,
    rLIMIT_HH := MS_DTRO_HH,
    rLIMIT_HI := MS_DTRO_HI,
    tDELAY_HH := TD_DTRO_HH,
    tDELAY_HI := TD_DTRO_HI,
    bERROR := _w7,
    bFAULT := _w8); // BWTS.ALARM_TRO
DTRO_HH_P := ALARM_TRO_DEBAL_P.HH;
DTRO_HI_P := ALARM_TRO_DEBAL_P.HI;
TRO_PORT := SEL(TRO_CROSS, AIT_251, AIT_151);
TRO_STBD := SEL(NOT TRO_CROSS, AIT_251, AIT_151);
(* SEL(TRO01_SEL, AIT_251_F, AIT_151_F); result not used *)
(* SEL(TRO01_SEL, FALSE, FALSE); result not used *)
ALARM_TRO_STR(
    rTRO := TRO_STR,
    bTRIGGER := SST_S_04.COMPLETE,
    tSUPPRESS := MS_DTRO_STABLE,
    rLIMIT_HH := MS_DTRO_HH,
    rLIMIT_HI := MS_DTRO_HI,
    tDELAY_HH := TD_DTRO_HH,
    tDELAY_HI := TD_DTRO_HI,
    bERROR := _w9,
    bFAULT := _w10); // BWTS.ALARM_TRO
STRO_HH := ALARM_TRO_STR.HH;
STRO_HI := ALARM_TRO_STR.HI;
TRO_STR := SEL(TRO01_SEL, AIT_251, AIT_151);

END_PROGRAM

// Device/Application/Logic/0.ETC/LINE_UP
PROGRAM LINE_UP
VAR
END_VAR

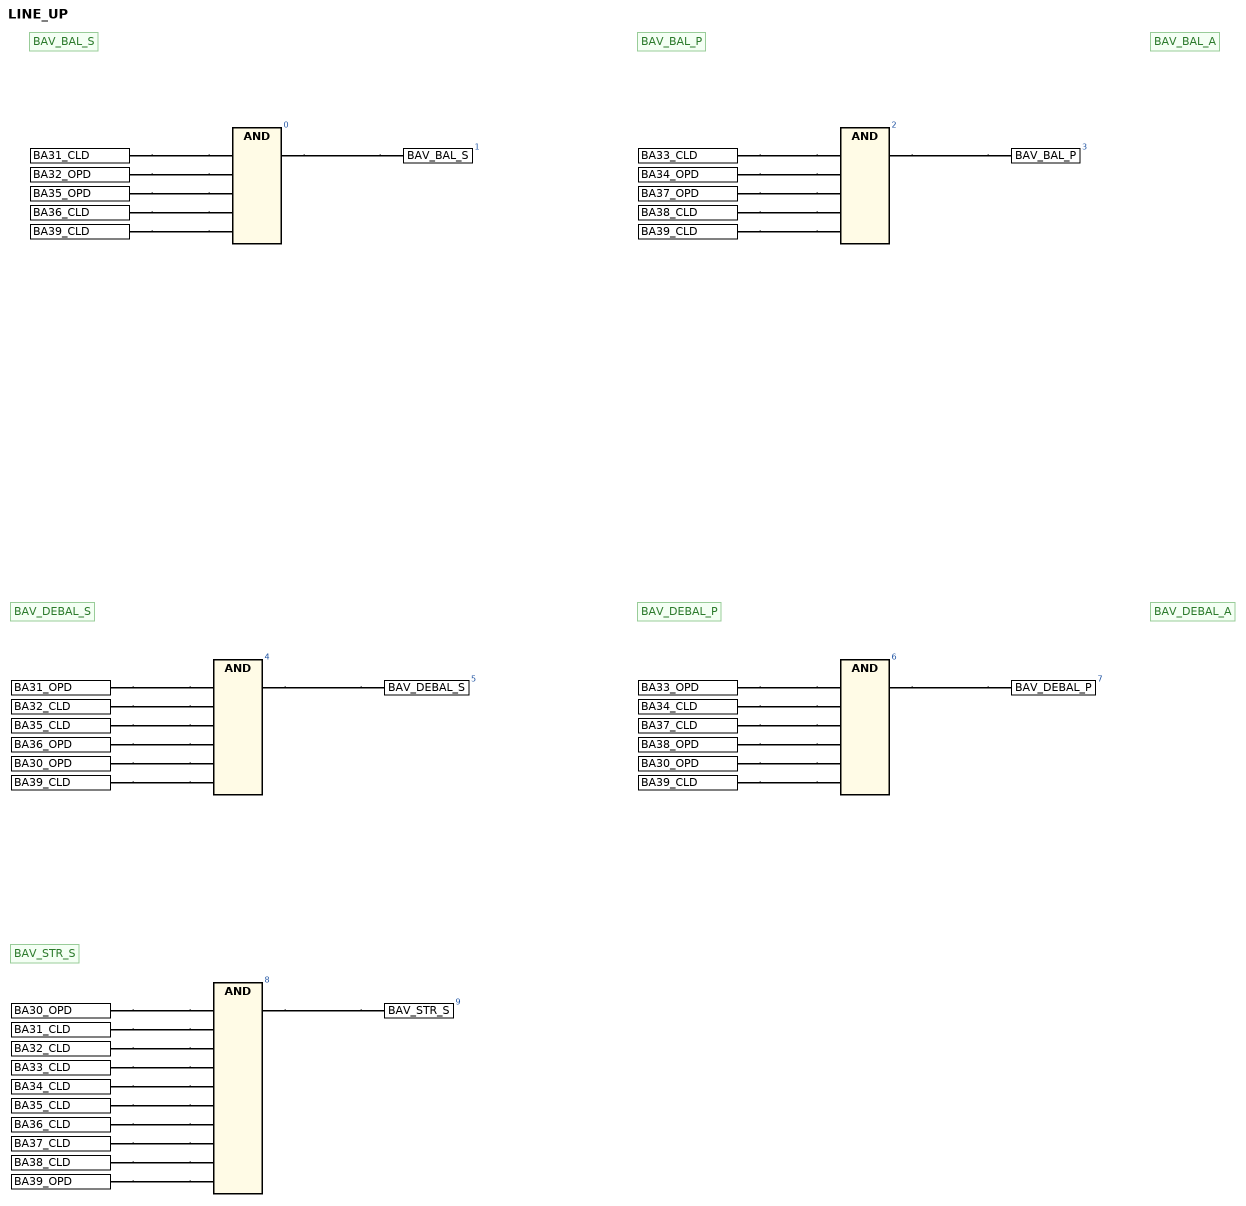
// BAV_BAL_S
BAV_BAL_S := BA31_CLD AND BA32_OPD AND BA35_OPD AND BA36_CLD AND BA39_CLD;
// BAV_BAL_P
// BAV_BAL_A
BAV_BAL_P := BA33_CLD AND BA34_OPD AND BA37_OPD AND BA38_CLD AND BA39_CLD;
// BAV_DEBAL_S
BAV_DEBAL_S := BA31_OPD AND BA32_CLD AND BA35_CLD AND BA36_OPD AND BA30_OPD AND BA39_CLD;
// BAV_DEBAL_P
// BAV_DEBAL_A
BAV_DEBAL_P := BA33_OPD AND BA34_CLD AND BA37_CLD AND BA38_OPD AND BA30_OPD AND BA39_CLD;
// BAV_STR_S
BAV_STR_S := BA30_OPD AND BA31_CLD AND BA32_CLD AND BA33_CLD AND BA34_CLD AND BA35_CLD AND BA36_CLD AND BA37_CLD AND BA38_CLD AND BA39_OPD;

END_PROGRAM

// Device/Application/Logic/0.ETC/MAINTENANCE_AND_DISABLE
PROGRAM MAINTENANCE_AND_DISABLE
VAR
	RS_0: RS;
	RS_1: RS;
	RS_2: RS;
	RS_3: RS;
	RS_4: RS;
	RS_5: RS;
	RS_6: RS;
	RS_7: RS;
END_VAR

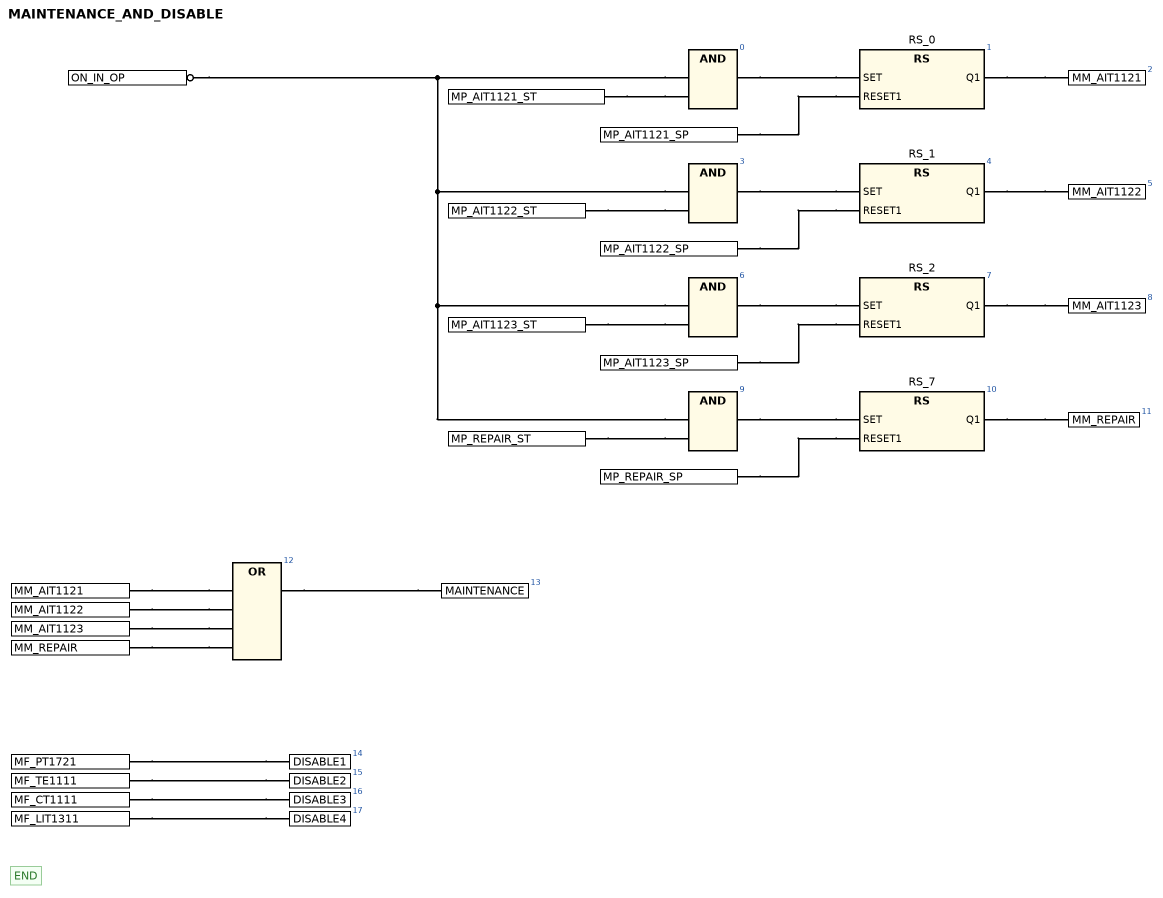
RS_0(SET := NOT ON_IN_OP AND MP_AIT1121_ST, RESET1 := MP_AIT1121_SP); // RS
MM_AIT1121 := RS_0.Q1;
RS_1(SET := NOT ON_IN_OP AND MP_AIT1122_ST, RESET1 := MP_AIT1122_SP); // RS
MM_AIT1122 := RS_1.Q1;
RS_2(SET := NOT ON_IN_OP AND MP_AIT1123_ST, RESET1 := MP_AIT1123_SP); // RS
MM_AIT1123 := RS_2.Q1;
RS_7(SET := NOT ON_IN_OP AND MP_REPAIR_ST, RESET1 := MP_REPAIR_SP); // RS
MM_REPAIR := RS_7.Q1;
MAINTENANCE := MM_AIT1121 OR MM_AIT1122 OR MM_AIT1123 OR MM_REPAIR;
DISABLE1 := MF_PT1721;
DISABLE2 := MF_TE1111;
DISABLE3 := MF_CT1111;
// END
DISABLE4 := MF_LIT1311;

END_PROGRAM

// Device/Application/Logic/0.ETC/RF_CC
PROGRAM RF_CC
VAR
	CCSS_RF142A: BWTS.CCSS;
	CCSS_RF142B: BWTS.CCSS;
	CCSS_RF142C: BWTS.CCSS;
END_VAR

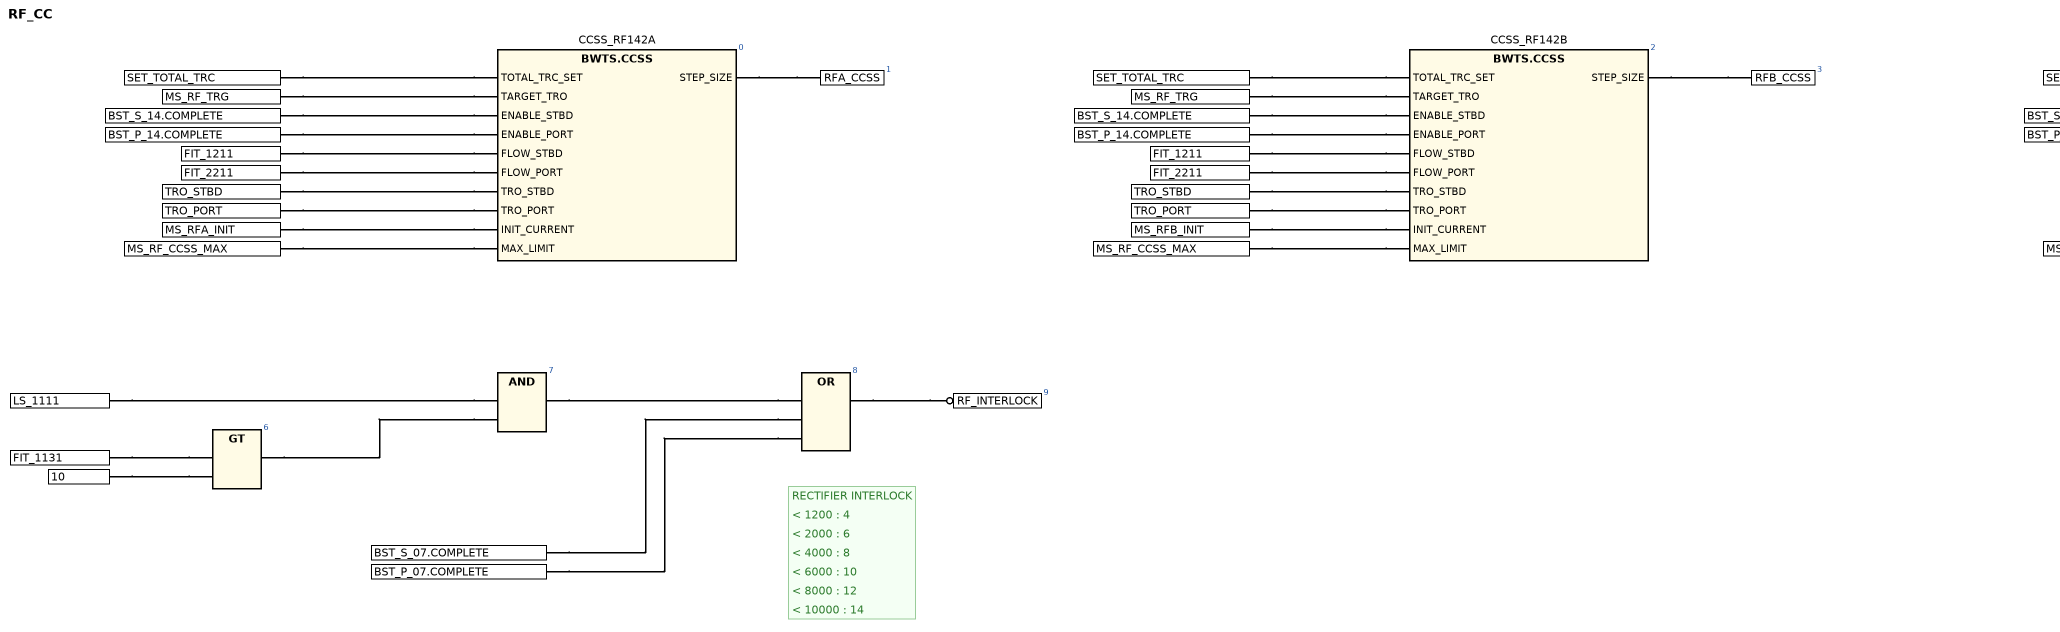
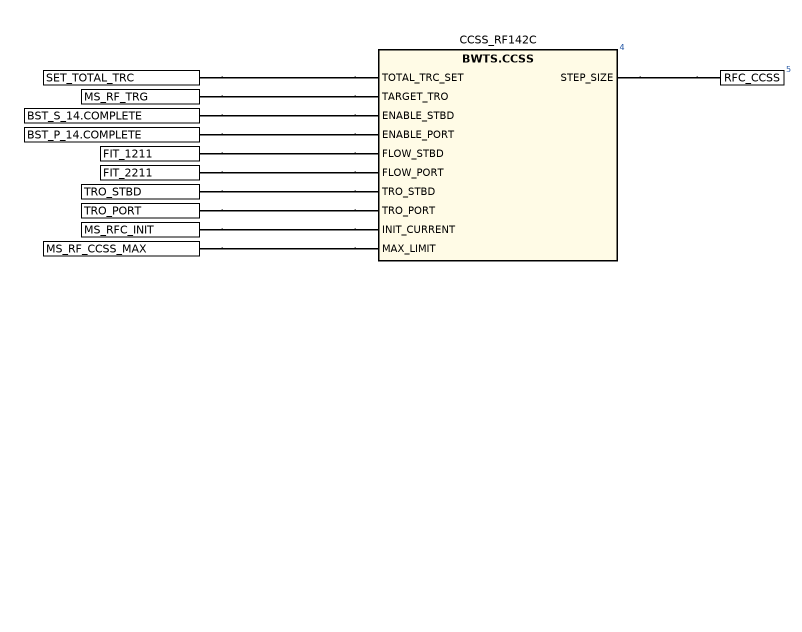
CCSS_RF142A(
    TOTAL_TRC_SET := SET_TOTAL_TRC,
    TARGET_TRO := MS_RF_TRG,
    ENABLE_STBD := BST_S_14.COMPLETE,
    ENABLE_PORT := BST_P_14.COMPLETE,
    FLOW_STBD := FIT_1211,
    FLOW_PORT := FIT_2211,
    TRO_STBD := TRO_STBD,
    TRO_PORT := TRO_PORT,
    INIT_CURRENT := MS_RFA_INIT,
    MAX_LIMIT := MS_RF_CCSS_MAX); // BWTS.CCSS
RFA_CCSS := CCSS_RF142A.STEP_SIZE;
CCSS_RF142B(
    TOTAL_TRC_SET := SET_TOTAL_TRC,
    TARGET_TRO := MS_RF_TRG,
    ENABLE_STBD := BST_S_14.COMPLETE,
    ENABLE_PORT := BST_P_14.COMPLETE,
    FLOW_STBD := FIT_1211,
    FLOW_PORT := FIT_2211,
    TRO_STBD := TRO_STBD,
    TRO_PORT := TRO_PORT,
    INIT_CURRENT := MS_RFB_INIT,
    MAX_LIMIT := MS_RF_CCSS_MAX); // BWTS.CCSS
RFB_CCSS := CCSS_RF142B.STEP_SIZE;
CCSS_RF142C(
    TOTAL_TRC_SET := SET_TOTAL_TRC,
    TARGET_TRO := MS_RF_TRG,
    ENABLE_STBD := BST_S_14.COMPLETE,
    ENABLE_PORT := BST_P_14.COMPLETE,
    FLOW_STBD := FIT_1211,
    FLOW_PORT := FIT_2211,
    TRO_STBD := TRO_STBD,
    TRO_PORT := TRO_PORT,
    INIT_CURRENT := MS_RFC_INIT,
    MAX_LIMIT := MS_RF_CCSS_MAX); // BWTS.CCSS
RFC_CCSS := CCSS_RF142C.STEP_SIZE;
// RECTIFIER INTERLOCK
// < 1200 : 4
// < 2000 : 6
// < 4000 : 8
// < 6000 : 10
// < 8000 : 12
// < 10000 : 14
RF_INTERLOCK := NOT (LS_1111 AND FIT_1131 > 10 OR BST_S_07.COMPLETE OR BST_P_07.COMPLETE);

END_PROGRAM

// Device/Application/Logic/0.ETC/SELECTION
PROGRAM SELECTION
VAR
	RS_0: RS; //BLOWER SELECTION
	RS_1: RS; //SWFP SELECATION
	RS_2: RS; //RFC DISABLE
	RS_3: RS; //RFA DISABLE
	RS_4: RS; //RFB DISABLE
	RS_5: RS; //NU CROSS
	RS_6: RS; //NU SELECTION
	RS_7: RS; //GSP SELECTION
	RS_10: RS; //TRO SELECTION
	RS_SEA_EN: RS;
	RS_SEA_EN_S: RS;
	RS_SEA_EN_P: RS;
	RS_CIR_EN_S: RS;
	RS_CIR_EN_P: RS;
	RS_TRO_CROSS: RS;
	TP_0: TP;
END_VAR
VAR // added by the converter: edge detectors and wires of the graphical bodies
    _w1, _w2, _w3, _w4, _w5, _w6, _w7 : ANY;
END_VAR

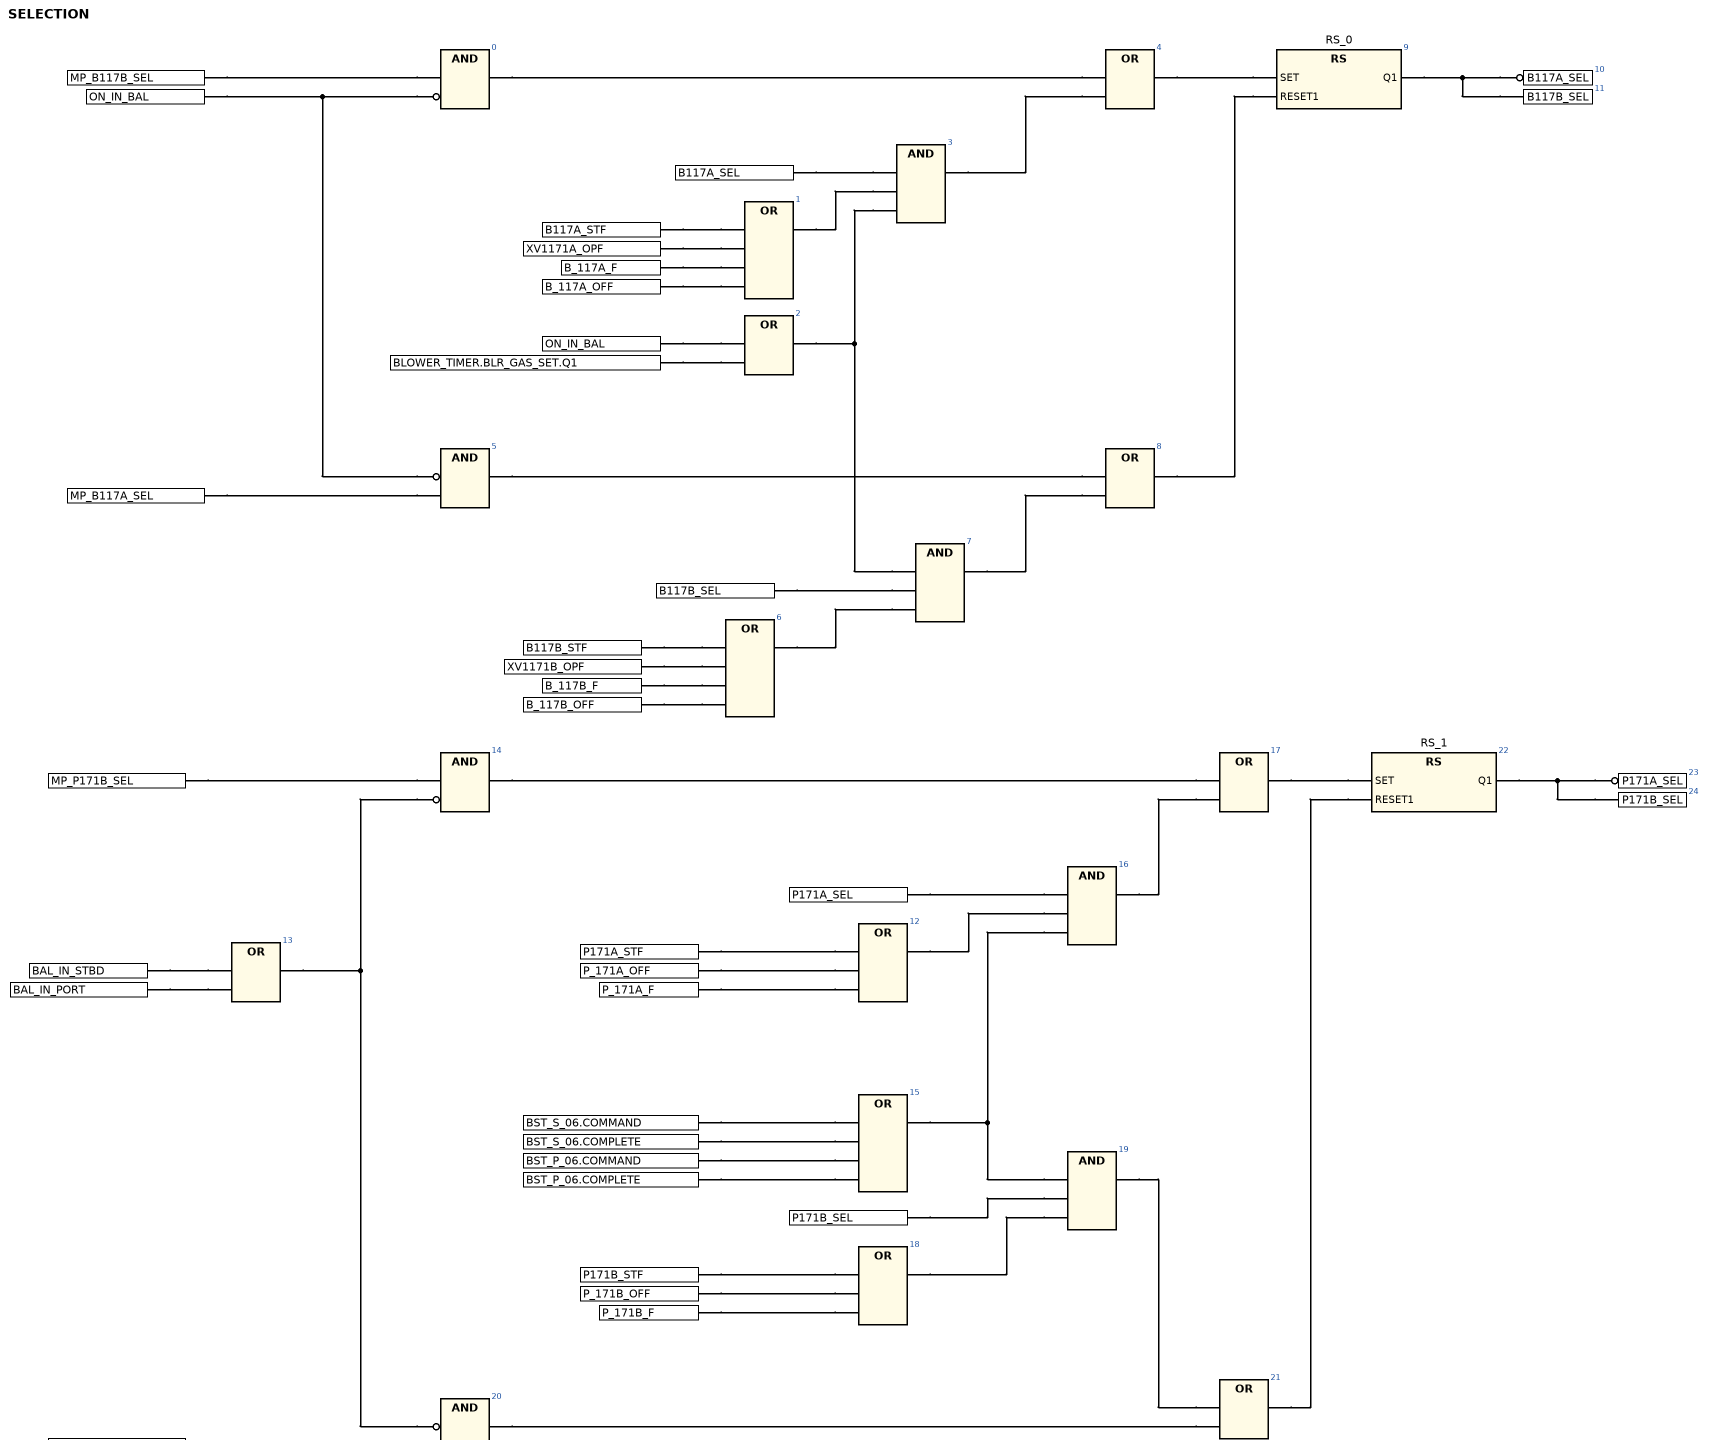
